# B&R Automation Studio project Soiled_PLC (part 9)

### CAN.typ
```iecst
TYPE
	WET_CAN : 	STRUCT
		ControlSignals : USINT;
		ControlSignals2 : USINT;
		Category : UINT;
		Customer : UINT;
		Weight : UINT;
	END_STRUCT;
	DRY_CAN : 	STRUCT
		ControlSignals : USINT;
		ControlByte2 : USINT;
		Category : UDINT;
		Weight : UINT;
	END_STRUCT;
	DRY_CAN1 : 	STRUCT
		CustomerCode : UDINT;
		BatchCode : UDINT;
	END_STRUCT;
	DRYCAN_comm_typ : 	STRUCT
		ReadFrame : DRY_CAN;
		WriteFrame : DRY_CAN;
		WriteFrame1 : DRY_CAN1;
		EventRead : BOOL;
		EventWrite : BOOL;
		EventWrite1 : BOOL;
	END_STRUCT;
	CAN_Vars : 	STRUCT
		StrobeComplete : BOOL;
		BagReady : BOOL;
		BatchCode : UINT;
		Category : UDINT;
		Customer : UDINT;
		Destination : UINT;
		DropLoad : BOOL;
		DoubleLoad : BOOL;
		Drier1Loading : BOOL;
		Drier2Loading : BOOL;
		Drier1Unloading : BOOL;
		Drier2Unloading : BOOL;
		FaultNumber : USINT;
		Live : BOOL;
		LiveTime : UINT;
		LoadDropped : BOOL;
		LoadFinished : BOOL;
		MachineID : UINT;
		Program : UINT;
		PressShift : BOOL;
		ReadyToLoad : BOOL;
		SP1 : UINT;
		SP2 : UINT;
		SP3 : UINT;
		Transfer : BOOL;
		UnloadFinished : BOOL;
		Weight : UINT;
		BatchID : UDINT;
		Batch_QtyRemaining : UINT;
		LoadRecieved : BOOL;
		Unloading : BOOL;
		Batchpart : ARRAY[0..7]OF Batchpart_typ;
		Batchpart_wgt : ARRAY[0..9]OF UINT;
	END_STRUCT;
	Batchpart_typ : 	STRUCT
		Wgt : UINT;
		Customer : UDINT;
	END_STRUCT;
	Comm_typ : 	STRUCT
		StrobeComplete : BOOL;
		BagReady : BOOL;
		BatchCode : UINT;
		Category : UDINT;
		Customer : UDINT;
		Destination : UINT;
		DropLoad : BOOL;
		DoubleLoad : BOOL;
		Live : BOOL;
		LiveTime : UINT;
		LoadDropped : BOOL;
		LoadFinished : BOOL;
		Program : UINT;
		ReadyToLoad : BOOL;
		UnloadFinished : BOOL;
		Weight : UINT;
		BatchID : UDINT;
		Batch_QtyRemaining : UINT;
		LoadRecieved : BOOL;
		Unloading : BOOL;
		Batchpart : ARRAY[0..7]OF Batchpart_typ;
		Batchpart_wgt : ARRAY[0..9]OF UINT;
		Count : UINT;
		Bid : UDINT; (**Internal use only pass bid ID>*)
		TimeStamp : DATE_AND_TIME; (**Internal use only*)
		Transfer : BOOL;
	END_STRUCT;
END_TYPE
```

### Program Logical/Sequences/200ms/CAN/can (IEC, version 2.00.0) - *DRY CAN

#### can.var
```iecst
VAR RETAIN
	CAN_enable : BOOL;
END_VAR
VAR
	CANdftab_01 : CANdftab;
	CANOK : BOOL;
	CANopen_01 : CANopen;
	CANrwtab_01 : CANrwtab;
	data_adr : UDINT;
	DOInfo : DatObjInfo;
	error_var : UDINT;
	LastError : UINT;
	n : UINT;
	MAX_CAN_CONNS : UINT;
	CAN_DRY_Send : ARRAY[0..19] OF DRYCAN_comm_typ;
	x : UINT;
END_VAR
```

#### can.ab
```automation-basic
;CAN Bus data exchange with CBW

;--------------------------------------------------------
;Version 1.00 02/11/2009 D.J. First Issue
;Version 2.00 22/011/2011 D.J. Weight Calculation now here
;--------------------------------------------------------

PROGRAM _INIT

CAN_enable = 1
MAX_CAN_CONNS = 6

LOOP n = 1 TO MAX_CAN_CONNS DO
	CAN_DRY_Send[n].EventRead = 0
	CAN_DRY_Send[n].EventWrite = 0
	CAN_DRY_Send[n].EventWrite1 = 0
ENDLOOP

CANopen_01.enable		= CAN_enable
CANopen_01.baud_rate	= 25					;Define baud rate - 250 kbit/s
CANopen_01.cob_anz		= 100      				;Define number of link objects
CANopen_01.error_adr	= ADR(error_var)		;Define address for error output
CANopen_01.device		= ADR("SS1.IF2")	    ;Define number of device
CANopen_01.info			= 0

CANopen_01 FUB CANopen()						;Initiate CANopen

IF CANopen_01.status=0 THEN						;Check error level

	DOInfo.enable = 1
	DOInfo.pName  = "can_cmd"

	DOInfo FUB DatObjInfo()

	IF (DOInfo.status = 0) THEN

		data_adr					= DOInfo.pDatObjMem
		CANdftab_01.enable			= 1
		CANdftab_01.us_ident 		= CANopen_01.us_ident	;Set us_id
		CANdftab_01.table_adr		= data_adr				;Define address of data object
		CANdftab_01.tab_num			= UINT(DOInfo.len / 72)	;Define number of values

		CANdftab_01 FUB CANdftab()    						;Initiate CANdftab

		IF CANdftab_01.status = 0 THEN
			LOOP n = 1 TO MAX_CAN_CONNS DO
				CAN_DRY_Send[n].WriteFrame.ControlSignals.0 = 1 // Set CAN Live
			ENDLOOP
			CANOK = TRUE
		ENDIF
	ENDIF
ENDIF

END_PROGRAM

PROGRAM _CYCLIC

IF CANOK THEN

	;----------------
	;Set Write values
	;---------------
	LOOP n = 3 TO MAX_CAN_CONNS DO
		CAN_DRY_Send[n].WriteFrame.ControlSignals.1 = CAN[n].BagReady
		CAN_DRY_Send[n].WriteFrame.Category			= CAN[n].Category
		CAN_DRY_Send[n].WriteFrame.Weight			= CAN[n].Weight
		CAN_DRY_Send[n].WriteFrame1.CustomerCode	= CAN[n].Customer
		CAN_DRY_Send[n].WriteFrame1.BatchCode		= CAN[n].BatchID
		CAN_DRY_Send[n].EventWrite = 1
		CAN_DRY_Send[n].EventWrite1 = 1
	ENDLOOP

	;-----------------
	;Service CAN table
	;-----------------
	IF CANdftab_01.status=0 THEN						(*check error level*)
		CANrwtab_01.enable		= 1
		CANrwtab_01.tab_ident	= CANdftab_01.tab_ident (*define tab_id*)
		CANrwtab_01 FUB CANrwtab()						(*initiate CANrwtab*)
		LastError = CANrwtab_01.status
	ENDIF

;	;----------------------------------
		;	;Check for incomming data from CBW1
		;	;----------------------------------
	LOOP n = 3 TO MAX_CAN_CONNS DO

		IF (CAN_DRY_Send[n].EventRead > 0)THEN
			CAN_DRY_Send[n].EventRead = 0

			CAN[n].Live 		  = CAN_DRY_Send[n].ReadFrame.ControlSignals.0
			CAN[n].DropLoad 	  = CAN_DRY_Send[n].ReadFrame.ControlSignals.1
			CAN[n].LoadDropped    = CAN_DRY_Send[n].ReadFrame.ControlSignals.2
			IF CAN[n].Live THEN
				CAN[n].LiveTime = 50	;5 seconds
			ENDIF
		ENDIF
		;~~~~~~~~~~~~~~~~~~~~~~~~~~~~~~~~~~~~~~~~~~~~~~~~
		;-------------------
		;CAN Live / Presence
		;-------------------
		IF (CAN[n].LiveTime > 0) THEN
			CAN[n].LiveTime = (CAN[n].LiveTime - 1)
		ENDIF
		CAN[n].Live = (CAN[n].LiveTime <> 0)

	ENDLOOP

ENDIF
END_PROGRAM
```

### Data object Logical/Sequences/200ms/CAN/can_cmd_wet (Simple) - *WET CAN I

#### can_cmd.dat
```
;-----------------
;CAN Command Table
;-----------------

;         1234567890123456789012345678901   1234567890123456789012345678901
00000121,"CAN_Drv2:ReadFrame1            ","CAN_Drv2:EventRead1            ",$00000000
00000120,"CAN_Drv2:WriteFrame1           ","CAN_Drv2:EventWrite1           ",$00000001

00000131,"CAN_Drv2:ReadFrame2            ","CAN_Drv2:EventRead2            ",$00000000
00000130,"CAN_Drv2:WriteFrame2           ","CAN_Drv2:EventWrite2           ",$00000001

; CAN ADR  Variable Name 31 Chrs             Event Variable 31 Chrs           Read = 0 Write = 1
```

- Program Logical/Sequences/200ms/CAN/CAN_Live (IEC) - * CAN Live status 1-32 to TrackView (no source held here)

### Data object Logical/Sequences/200ms/CAN/can1_cmd (Simple, version 1.00.0) - * Powertrans 1 & 2

#### can_cmd.dat
```
;-----------------
;CAN Command Table
;-----------------

;         1234567890123456789012345678901   1234567890123456789012345678901
00000251,"can_drv1:ReadFrame1            ","can_drv1:EventRead1            ",$00000000
00000241,"can_drv1:WriteFrame1           ","can_drv1:EventWrite1           ",$00000001
;123456789123456789123456789123456789123456789123456789123456789123456789
;00000121,"can_drv1:ReadFrame2            ","can_drv1:EventRead2            ",$00000000
;00000120,"can_drv1:WriteFrame2           ","can_drv1:EventWrite2           ",$00000001

;00000141,"ReadFrame3                     ","EventRead3                     ",$00000000
;00000140,"WriteFrame3                    ","EventWrite3                    ",$00000001
;   |          |                                 |                               |
; CAN ADR  Variable Name 31 Chrs             Event Variable 31 Chrs           Read = 0 Write = 1
```

### Program Logical/Sequences/200ms/CAN/can_drv1 (IEC) - * PowerTrans 1 SDC2

#### can_drv2.var
```iecst
VAR RETAIN
	CAN_enable : BOOL;
	ReadFrame1 : WET_CAN;
	EventRead1 : BOOL;
	EventWrite1 : BOOL;
	LastError : UINT;
	n : UINT;
	CANOK : BOOL;
	WriteFrame1 : WET_CAN;
	EventWrite2 : BOOL;
END_VAR
VAR
	ReadFrame2 : WET_CAN;
	EventRead2 : BOOL;
	WriteFrame2 : WET_CAN;
	CANopen_01 : CANopen;
	DOInfo : DatObjInfo;
	CANdftab_01 : CANdftab;
	error_var : UDINT;
	data_adr : UDINT;
	CANrwtab_01 : CANrwtab;
	TEST : BOOL;
END_VAR
```

#### can_drv2Cyclic.ab
```automation-basic
PROGRAM _CYCLIC
;----------------------------------------
;Version 1.00 08/02/2005 D.J. First Issue
;----------------------------------------

IF CANOK THEN

	;----------------
	;Set Write values
	;----------------

	;Powertrans 1
	IF CAN[1].BagReady THEN
		WriteFrame1.ControlSignals = BIT_SET(WriteFrame1.ControlSignals, 1)
	ELSE
		WriteFrame1.ControlSignals = BIT_CLR(WriteFrame1.ControlSignals, 1)
	ENDIF
   IF CAN[1].LoadFinished = TRUE THEN
			WriteFrame1.ControlSignals = BIT_SET(WriteFrame1.ControlSignals, 2)
	ELSE
			WriteFrame1.ControlSignals = BIT_CLR(WriteFrame1.ControlSignals, 2)
	ENDIF
	//WriteFrame1.Destination = 0
	WriteFrame1.Category 	= UINT(CAN[1].Category)
	WriteFrame1.Customer    = UINT(CAN[1].Customer)
	WriteFrame1.Weight      = CAN[1].Weight

	;Write to Machine1
	EventWrite1 = TRUE

	;Powertrans 2
	IF CAN[2].BagReady THEN
		WriteFrame2.ControlSignals = BIT_SET(WriteFrame2.ControlSignals, 1)
	ELSE
		WriteFrame2.ControlSignals = BIT_CLR(WriteFrame2.ControlSignals, 1)
	ENDIF
	;IF CAN[2].DoubleLoad THEN
	;	WriteFrame2.ControlSignals = BIT_SET(WriteFrame2.ControlSignals, 2)
	;ELSE
	;	WriteFrame2.ControlSignals = BIT_CLR(WriteFrame2.ControlSignals, 2)
	;ENDIF
	//WriteFrame2.Destination = 0
	WriteFrame2.Category 	= UINT(CAN[2].Category)
	WriteFrame2.Customer    = UINT(CAN[2].Customer)
	WriteFrame2.Weight      = CAN[2].Weight

	;Write to Machine2
	EventWrite2 = TRUE

	;-----------------
	;Service CAN table
	;-----------------

	IF CANdftab_01.status=0 THEN						(*check error level*)
		CANrwtab_01.enable		= 1
		CANrwtab_01.tab_ident	= CANdftab_01.tab_ident (*define tab_id*)
		CANrwtab_01 FUB CANrwtab()						(*initiate CANrwtab*)
		LastError = CANrwtab_01.status
	ENDIF

	;----------------------------------
	;Check for incomming data from CBW1
	;----------------------------------

	;Powertrans 1
	IF EventRead1 THEN

		EventRead1 = FALSE

		CAN[1].Live 		  = BIT_TST(ReadFrame1.ControlSignals,0)
		CAN[1].ReadyToLoad 	  = BIT_TST(ReadFrame1.ControlSignals,1)
        CAN[1].DropLoad           =  BIT_TST(ReadFrame1.ControlSignals,2)
		CAN[1].LoadDropped    = BIT_TST(ReadFrame1.ControlSignals,3)

		IF CAN[1].Live THEN
			CAN[1].LiveTime = 50	;5 seconds
		ENDIF

	ENDIF

	;----------------------------------
	;Check for incomming data from CBW2
	;----------------------------------

	;Powertrans 2
	IF EventRead2 THEN

		EventRead2 = FALSE

		CAN[2].Live 		  = BIT_TST(ReadFrame2.ControlSignals,0)
		CAN[2].DropLoad 	  = BIT_TST(ReadFrame2.ControlSignals,1)
		CAN[2].LoadDropped    = BIT_TST(ReadFrame2.ControlSignals,2)

		IF CAN[2].Live THEN
			CAN[2].LiveTime = 50	;5 seconds
		ENDIF

	ENDIF

	;-------------------
	;CAN Live / Presence
	;-------------------

	LOOP n = 1 TO 2 DO

		IF (CAN[n].LiveTime > 0) THEN
			CAN[n].LiveTime = (CAN[n].LiveTime - 1)
		ENDIF

		CAN[n].Live = (CAN[n].LiveTime <> 0)

	ENDLOOP

ENDIF
END_PROGRAM
```

#### can_drv2Init.ab
```automation-basic
PROGRAM _INIT
	(* init program *)

CAN_enable = 1
EventWrite1 = 0									;Reset CAN data table WRITE event
EventRead1 = 0  								;Reset CAN data table READ event
;EventWrite2 = 0								;Reset CAN data table WRITE event
;EventRead2 = 0  								;Reset CAN data table READ event
;EventWrite3 = 0								;Reset CAN data table WRITE event
;EventRead3 = 0  							    ;Reset CAN data table READ event

CANopen_01.enable		= CAN_enable
CANopen_01.baud_rate	= 25					;Define baud rate - 250 kbit/s
CANopen_01.cob_anz		= 100      				;Define number of link objects
CANopen_01.error_adr	= ADR(error_var)		;Define address for error output
CANopen_01.device		= ADR("SS1.IF1")	;Define number of device
CANopen_01.info			= 0

CANopen_01 FUB CANopen()						;Initiate CANopen

IF CANopen_01.status=0 THEN						;Check error level

	DOInfo.enable = 1
	DOInfo.pName  = "can1_cmd"

	DOInfo FUB DatObjInfo()

	IF (DOInfo.status = 0) THEN

		data_adr					= DOInfo.pDatObjMem
		CANdftab_01.enable			= 1
		CANdftab_01.us_ident 		= CANopen_01.us_ident	;Set us_id
		CANdftab_01.table_adr		= data_adr				;Define address of data object
		CANdftab_01.tab_num			= UINT(DOInfo.len / 72)	;Define number of values

		CANdftab_01 FUB CANdftab()    						;Initiate CANdftab

		IF CANdftab_01.status = 0 THEN
			WriteFrame1.ControlSignals = BIT_SET(WriteFrame1.ControlSignals,0);Set Live Signal
			WriteFrame2.ControlSignals = BIT_SET(WriteFrame2.ControlSignals,0)
			;WriteFrame3.ControlSignals = BIT_SET(WriteFrame3.ControlSignals,0)
			CANOK = TRUE
		ENDIF

	ENDIF

ENDIF
END_PROGRAM
```

### Program Logical/Sequences/200ms/CAN/can_drv2 (IEC, version 1.00.0) - * PowerTrans 1 SDC2

#### can_drv2Cyclic.ab
```automation-basic
PROGRAM _CYCLIC
;----------------------------------------
;Version 1.00 08/02/2005 D.J. First Issue
;----------------------------------------

IF CANOK THEN

	;----------------
	;Set Write values
	;----------------

	;Powertrans 1
	IF CAN[2].BagReady THEN
		WriteFrame2.ControlSignals = BIT_SET(WriteFrame2.ControlSignals, 1)
	ELSE
		WriteFrame2.ControlSignals = BIT_CLR(WriteFrame2.ControlSignals, 1)
	ENDIF
 IF CAN[2].LoadFinished = TRUE THEN
			WriteFrame2.ControlSignals = BIT_SET(WriteFrame2.ControlSignals, 2)
	ELSE
			WriteFrame2.ControlSignals = BIT_CLR(WriteFrame2.ControlSignals, 2)
	ENDIF
	//WriteFrame1.Destination = 0
	WriteFrame2.Category 	= UINT(CAN[2].Category)
	WriteFrame2.Customer    = UINT(CAN[2].Customer)
	WriteFrame2.Weight      = CAN[2].Weight

	;Write to Machine1
	EventWrite2 = TRUE

	//WriteFrame2.Destination = 0
	WriteFrame2.Category 	= UINT(CAN[2].Category)
	WriteFrame2.Customer    = UINT(CAN[2].Customer)
	WriteFrame2.Weight      = CAN[2].Weight

	;Write to Machine2
	EventWrite2 = TRUE

	;-----------------
	;Service CAN table
	;-----------------

	IF CANdftab_01.status=0 THEN						(*check error level*)
		CANrwtab_01.enable		= 1
		CANrwtab_01.tab_ident	= CANdftab_01.tab_ident (*define tab_id*)
		CANrwtab_01 FUB CANrwtab()						(*initiate CANrwtab*)
		LastError = CANrwtab_01.status
	ENDIF

	;----------------------------------
	;Check for incomming data from CBW1
	;----------------------------------

	;Powertrans 1
	IF EventRead2 THEN

		EventRead2 = FALSE

		CAN[2].Live 		          = BIT_TST(ReadFrame2.ControlSignals,0)
		CAN[2].ReadyToLoad	  = BIT_TST(ReadFrame2.ControlSignals,1)
		CAN[2].DropLoad          = BIT_TST(ReadFrame2.ControlSignals,2)
		CAN[2].LoadDropped    = BIT_TST(ReadFrame2.ControlSignals,3)

		IF CAN[2].Live THEN
			CAN[2].LiveTime = 50	;5 seconds
		ENDIF

	ENDIF

	;----------------------------------
	;Check for incomming data from CBW2
	;----------------------------------

	;-------------------
	;CAN Live / Presence
	;-------------------

	LOOP n = 1 TO 2 DO

		IF (CAN[n].LiveTime > 0) THEN
			CAN[n].LiveTime = (CAN[n].LiveTime - 1)
		ENDIF

		CAN[n].Live = (CAN[n].LiveTime <> 0)

	ENDLOOP

ENDIF
END_PROGRAM
```

#### can_drv2Init.ab
```automation-basic
PROGRAM _INIT
	(* init program *)

CAN_enable = 1
EventWrite1 = 0									;Reset CAN data table WRITE event
EventRead1 = 0  								;Reset CAN data table READ event
;EventWrite2 = 0								;Reset CAN data table WRITE event
;EventRead2 = 0  								;Reset CAN data table READ event
;EventWrite3 = 0								;Reset CAN data table WRITE event
;EventRead3 = 0  							    ;Reset CAN data table READ event

CANopen_01.enable		= CAN_enable
CANopen_01.baud_rate	= 25					;Define baud rate - 250 kbit/s
CANopen_01.cob_anz		= 100      				;Define number of link objects
CANopen_01.error_adr	= ADR(error_var)		;Define address for error output
CANopen_01.device		= ADR("SS1.IF2")	;Define number of device
CANopen_01.info			= 0

CANopen_01 FUB CANopen()						;Initiate CANopen

IF CANopen_01.status=0 THEN						;Check error level

	DOInfo.enable = 1
	DOInfo.pName  = "can2_cmd"

	DOInfo FUB DatObjInfo()

	IF (DOInfo.status = 0) THEN

		data_adr					= DOInfo.pDatObjMem
		CANdftab_01.enable			= 1
		CANdftab_01.us_ident 		= CANopen_01.us_ident	;Set us_id
		CANdftab_01.table_adr		= data_adr				;Define address of data object
		CANdftab_01.tab_num			= UINT(DOInfo.len / 72)	;Define number of values

		CANdftab_01 FUB CANdftab()    						;Initiate CANdftab

		IF CANdftab_01.status = 0 THEN
			WriteFrame1.ControlSignals = BIT_SET(WriteFrame1.ControlSignals,0);Set Live Signal
			WriteFrame2.ControlSignals = BIT_SET(WriteFrame2.ControlSignals,0)
			;WriteFrame3.ControlSignals = BIT_SET(WriteFrame3.ControlSignals,0)
			CANOK = TRUE
		ENDIF

	ENDIF

ENDIF
END_PROGRAM
```

### Program Logical/Sequences/200ms/CAN/can_dis (IEC)

#### can_dis.var
```iecst
VAR RETAIN
	CAN_enable : BOOL;
	LastError : UINT;
	n : UINT;
	CANOK : BOOL;
END_VAR
VAR
	CANopen_01 : CANopen;
	DOInfo : DatObjInfo;
	CANdftab_01 : CANdftab;
	error_var : UDINT;
	data_adr : UDINT;
	CANrwtab_01 : CANrwtab;
	DisplayWrite1 : BOOL;
	DisplayRead1 : BOOL;
	DisplayCat : ARRAY[0..32] OF USINT;
	DisplayWgt : ARRAY[0..16] OF UINT;
	DisplayCus : ARRAY[0..32] OF USINT;
	Display : ARRAY[0..87] OF UINT;
	Data : WriteDisplay;
	Reply : USINT;
	DisplayRXFrame5 : ReadDisplay;
	DisplayRXFrame4 : ReadDisplay;
	DisplayWrite4 : BOOL;
	DisplayTXFrame1 : WriteDisplay;
	DisplayWrite5 : BOOL;
	DisplayTXFrame2 : WriteDisplay;
	x : UINT;
	DisplayWrite6 : BOOL;
	DisplayTXFrame3 : WriteDisplay;
	DisplayRead2 : BOOL;
	DisplayTXFrame4 : WriteDisplay;
	DisplayRead3 : BOOL;
	DisplayTXFrame5 : WriteDisplay;
	Dummy : UINT;
	DisplayRead4 : BOOL;
	DisplayRXFrame1 : ReadDisplay;
	DisplayTXFrame6 : WriteDisplay;
	DisplayRead5 : BOOL;
	DisplayRXFrame2 : ReadDisplay;
	DisplayRead6 : BOOL;
	DisplayRXFrame3 : ReadDisplay;
	StepsRequired : UINT;
	DisplayChrs : UINT;
	DisplayRXFrame6 : ReadDisplay;
	STEP : UINT;
	Wgt1s : UINT;
	DisplayWrite2 : BOOL;
	DisplayWrite3 : BOOL;
	Wgt10s : UINT;
	m : UINT;
	DisplayTXFrame7 : WriteDisplay;
	DisplayTXFrame8 : WriteDisplay;
	DisplayTXFrame9 : WriteDisplay;
	DisplayTXFrame10 : WriteDisplay;
	DisplayTXFrame11 : WriteDisplay;
	DisplayTXFrame12 : WriteDisplay;
	DisplayTXFrame13 : WriteDisplay;
	DisplayWrite7 : BOOL;
	DisplayWrite8 : BOOL;
	DisplayWrite9 : BOOL;
	DisplayWrite10 : BOOL;
	DisplayWrite11 : BOOL;
	DisplayWrite12 : BOOL;
	DisplayWrite13 : BOOL;
	DisplayWrite14 : BOOL;
	DisplayWrite15 : BOOL;
	DisplayWrite16 : BOOL;
	DisplayRead7 : BOOL;
	DisplayRead8 : BOOL;
	DisplayRead9 : BOOL;
	DisplayRead10 : BOOL;
	DisplayRead11 : BOOL;
	DisplayRead12 : BOOL;
	DisplayRead13 : BOOL;
	DisplayRead14 : BOOL;
	DisplayRead15 : BOOL;
	DisplayRead16 : BOOL;
	DisplayRXFrame7 : ReadDisplay;
	DisplayRXFrame8 : ReadDisplay;
	DisplayRXFrame9 : ReadDisplay;
	DisplayRXFrame10 : ReadDisplay;
	DisplayRXFrame11 : ReadDisplay;
	DisplayRXFrame12 : ReadDisplay;
	DisplayRXFrame13 : ReadDisplay;
	DisplayRXFrame14 : ReadDisplay;
	DisplayRXFrame15 : ReadDisplay;
	DisplayRXFrame16 : ReadDisplay;
	DisplayTXFrame14 : WriteDisplay;
	DisplayTXFrame15 : WriteDisplay;
	DisplayTXFrame16 : WriteDisplay;
	CatName : ARRAY[0..32] OF UINT;
	CusName : ARRAY[0..32] OF UINT;
END_VAR
```

#### can_disCyclic.ab
```automation-basic
PROGRAM _CYCLIC
;-----------------------------------------
;Revision 1.00 18/02/2002 D.J. First Issue
;-----------------------------------------

;2 * 20 or 2 * 40 chr VFD display

;Set D register where text for display is set E register for weight
DisplayChrs		= 80

;LOOP m = 1 TO 7 DO//16 DO
;
;
;	;memcpy(ADR(DisplayCat[m]),ADR(zzGetNamesData[m].CatName),16)
;;	memcpy(ADR(DisplayCus[m]),ADR(zzGetNamesData[m].CusName),16)
;
;ENDLOOP

LOOP x = 1 TO 7 DO//16 DO
	memcpy(ADR(DisplayCat[1]),ADR(zzGetNamesData[x].CatName),32);
	memcpy(ADR(DisplayCus[1]),ADR(zzGetNamesData[x].CusName),32)
	//Convert string to Wstring
	LOOP m = 1 TO 32 DO
		CatName[m] = UINT(DisplayCat[m])
		CusName[m] = UINT(DisplayCus[m])
	ENDLOOP

	DisplayWgt[x] = Bag[200 + x].Wgt

	memset(ADR(Display[0]) ,32,SIZEOF (Display))

	memcpy(ADR(Display[0]),ADR(CatName[1]),32)
	memcpy(ADR(Display[44]),ADR(CusName[1]),32)

	;As the weight value is a INT put into a UINT -0.1 = 65535
	;Display only if less than 500kg
	IF (DisplayWgt[x] < 5000) THEN
		DIS4(DisplayWgt[x],TRUE,Dummy,Wgt1s,Wgt10s,Dummy)
	ELSE
		Wgt1s 	= 0
		Wgt10s 	= 0
	ENDIF

	;Add Weight and goto next line
	Display[35] = $20 ;Space
	Display[36] = (48 + USINT(Wgt10s))
	Display[37] = (48 + USINT(Wgt1s))
	Display[38] = $6B 	;k
	Display[39] = $67 	;g
	Display[40] = $A	;Line Feed
	Display[41] = $D	;Carriage Return
	Display[42] = 0
	Display[43] = 0

	;Display[78] = $44	;D
	;Display[79] = $55	;U
	;Display[80] = $43	;C
	;Display[81] = $4B	;K
	;Display[82] = $45	;E
	;Display[83] = $52	;R

	;Cursor Off and Home
	IF (STEP = 0) THEN
		n = 0
		Data.Data[0] = $9B
		Data.Data[1] = $6C
		Data.Data[2] = $9B
		Data.Data[3] = $48
		Data.Data[4] = 0
		Data.Data[5] = 0
		Data.Data[6] = 0
		Data.Data[7] = 0
	ENDIF

	;Write text to the Display
	IF (STEP > 0) THEN
		Data.Data[0] = USINT(Display[0 + n])
		Data.Data[1] = USINT(Display[1 + n])
		Data.Data[2] = USINT(Display[2 + n])
		Data.Data[3] = USINT(Display[3 + n])
		Data.Data[4] = USINT(Display[4 + n])
		Data.Data[5] = USINT(Display[5 + n])
		Data.Data[6] = USINT(Display[6 + n])
		Data.Data[7] = USINT(Display[7 + n])
	ENDIF

	;Write to the CAN Frame For the Current Display
	IF (x = 1) THEN
		DisplayTXFrame1 = Data
	ELSE IF (x = 2) THEN
		DisplayTXFrame2 = Data
	ELSE IF (x = 3) THEN
		DisplayTXFrame3 = Data
	ELSE IF (x = 4) THEN
		DisplayTXFrame4 = Data
	ELSE IF (x = 5) THEN
		DisplayTXFrame5 = Data
	ELSE IF (x = 6) THEN
		DisplayTXFrame6 = Data
	ELSE IF (x = 7) THEN
		DisplayTXFrame7 = Data
	ELSE IF (x = 8) THEN
		DisplayTXFrame8 = Data
	ELSE IF (x = 9) THEN
		DisplayTXFrame9 = Data
	ELSE IF (x = 10) THEN
		DisplayTXFrame10 = Data
	ELSE IF (x = 11) THEN
		DisplayTXFrame11 = Data
	ELSE IF (x = 12) THEN
		DisplayTXFrame12 = Data
	ELSE IF (x = 13) THEN
		DisplayTXFrame13 = Data
	ELSE IF (x = 14) THEN
		DisplayTXFrame14 = Data
	ELSE IF (x = 15) THEN
		DisplayTXFrame15 = Data
	ELSE IF (x = 16) THEN
		DisplayTXFrame16 = Data
	ENDIF

ENDLOOP

IF (STEP > 0) THEN
	n = n + 8
ENDIF

STEP = STEP + 1

StepsRequired = ((DisplayChrs / 8) + 1) ;Steps = Total Chrs / 8 + 1
IF STEP > StepsRequired THEN
	STEP = 0
ENDIF

IF CANOK THEN

	;------------------------------------------------------
	;Configure the CAN write to CBW1 SDC1
	;------------------------------------------------------

	;Write to Displays
	DisplayWrite1 = TRUE
	;DisplayWrite2 = TRUE
	DisplayWrite3 = TRUE
	;DisplayWrite4 = TRUE
	DisplayWrite5 = TRUE
	;DisplayWrite6 = TRUE
	DisplayWrite7 = TRUE
	;DisplayWrite8 = TRUE
	;DisplayWrite9 = TRUE
	;DisplayWrite10 = TRUE
	;DisplayWrite11 = TRUE
	;DisplayWrite12 = TRUE
	;DisplayWrite13 = TRUE
	;DisplayWrite14 = TRUE
	;DisplayWrite15 = TRUE
	;DisplayWrite16 = TRUE

	;------------------------
	;Service CAN table
	;------------------------

	IF CANdftab_01.status=0 THEN						(*check error level*)
		CANrwtab_01.enable		= 1
		CANrwtab_01.tab_ident	= CANdftab_01.tab_ident (*define tab_id*)
		CANrwtab_01 FUB CANrwtab()						(*initiate CANrwtab*)
		LastError = CANrwtab_01.status
	ENDIF

	;-----------------
	;Read Display Data
	;-----------------
	IF DisplayRead1 THEN
		DisplayRead1 = FALSE
		Reply = DisplayRXFrame1.Data[1]
	ENDIF
	IF DisplayRead2 THEN
		DisplayRead2 = FALSE
		Reply = DisplayRXFrame2.Data[1]
	ENDIF
	IF DisplayRead3 THEN
		DisplayRead3 = FALSE
		Reply = DisplayRXFrame3.Data[1]
	ENDIF
	IF DisplayRead4 THEN
		DisplayRead4 = FALSE
		Reply = DisplayRXFrame4.Data[1]
	ENDIF
	IF DisplayRead5 THEN
		DisplayRead5 = FALSE
		Reply = DisplayRXFrame5.Data[1]
	ENDIF
	IF DisplayRead6 THEN
		DisplayRead6 = FALSE
		Reply = DisplayRXFrame6.Data[1]
	ENDIF
	IF DisplayRead7 THEN
		DisplayRead7 = FALSE
		Reply = DisplayRXFrame7.Data[1]
	ENDIF
	IF DisplayRead8 THEN
		DisplayRead8 = FALSE
		Reply = DisplayRXFrame8.Data[1]
	ENDIF
	IF DisplayRead9 THEN
		DisplayRead9 = FALSE
		Reply = DisplayRXFrame9.Data[1]
	ENDIF
	IF DisplayRead10 THEN
		DisplayRead10 = FALSE
		Reply = DisplayRXFrame10.Data[1]
	ENDIF
	IF DisplayRead11 THEN
		DisplayRead11 = FALSE
		Reply = DisplayRXFrame11.Data[1]
	ENDIF
	IF DisplayRead12 THEN
		DisplayRead12 = FALSE
		Reply = DisplayRXFrame12.Data[1]
	ENDIF
	IF DisplayRead13 THEN
		DisplayRead13 = FALSE
		Reply = DisplayRXFrame13.Data[1]
	ENDIF
	IF DisplayRead14 THEN
		DisplayRead14 = FALSE
		Reply = DisplayRXFrame14.Data[1]
	ENDIF
	IF DisplayRead15 THEN
		DisplayRead15 = FALSE
		Reply = DisplayRXFrame15.Data[1]
	ENDIF
	IF DisplayRead16 THEN
		DisplayRead16 = FALSE
		Reply = DisplayRXFrame16.Data[1]
	ENDIF

ENDIF

END_PROGRAM
```

#### can_disInit.ab
```automation-basic
PROGRAM _INIT
	(* init program *)

CAN_enable = 1
DisplayWrite1 = 0								;Reset CAN data table WRITE event
DisplayRead1 = 0  								;Reset CAN data table READ event
;EventWrite2 = 0								;Reset CAN data table WRITE event
;EventRead2 = 0  								;Reset CAN data table READ event
;EventWrite3 = 0								;Reset CAN data table WRITE event
;EventRead3 = 0  							    ;Reset CAN data table READ event

CANopen_01.enable		= CAN_enable
CANopen_01.baud_rate	= 25					;Define baud rate - 250 kbit/s
CANopen_01.cob_anz		= 100      				;Define number of link objects
CANopen_01.error_adr	= ADR(error_var)		;Define address for error output
CANopen_01.device		= ADR("SS1.IF2")		;Define number of device
CANopen_01.info			= 0

CANopen_01 FUB CANopen()						;Initiate CANopen

IF CANopen_01.status=0 THEN						;Check error level

	DOInfo.enable = 1
	DOInfo.pName  = "disp_cmd"

	DOInfo FUB DatObjInfo()

	IF (DOInfo.status = 0) THEN

		data_adr					= DOInfo.pDatObjMem
		CANdftab_01.enable			= 1
		CANdftab_01.us_ident 		= CANopen_01.us_ident	;Set us_id
		CANdftab_01.table_adr		= data_adr				;Define address of data object
		CANdftab_01.tab_num			= UINT(DOInfo.len / 72)	;Define number of values

		CANdftab_01 FUB CANdftab()    						;Initiate CANdftab

		IF CANdftab_01.status = 0 THEN
			CANOK = TRUE
		ENDIF

	ENDIF

ENDIF
END_PROGRAM
```

### Data object Logical/Sequences/200ms/CAN/can2_cmd (Simple)

#### disp_cmd.dat
```
;-----------------
;CAN Command Table
;-----------------

;         1234567890123456789012345678901   1234567890123456789012345678901
;CAN Node 11
00000251,"can_drv2:ReadFrame2            ","can_drv2:EventRead2            ",$00000000
00000241,"can_drv2:WriteFrame2           ","can_drv2:EventWrite2           ",$00000001

;   |          |                                 |                               |
; CAN ADR  Variable Name 31 Chrs             Event Variable 31 Chrs           Read = 0 Write = 1
```

### Package Logical/Sequences/200ms/Reports - Reports Variables

### Reports.typ
```iecst
TYPE
	Report : 	STRUCT
		Cat : UDINT;
		Cus : UDINT;
		Mis : UDINT;
		Bid : UDINT;
		Ur2 : UDINT;
		Prg : UINT;
		Wgt : UINT;
		Cnt : UINT;
		Stn : UINT;
		Mcn : UINT;
		Dst : UINT;
		Ur1 : UINT;
		Act : UINT;
		Rkg : UINT;
		TimeStamp : DATE_AND_TIME;
	END_STRUCT;
END_TYPE
```

### Reports.var
```iecst
VAR RETAIN
	ReportBuffer : ARRAY[0..199] OF Report;
	ReportLoading : ARRAY[0..60] OF Report;
	ReportUnloading : ARRAY[0..10] OF Report;
END_VAR
```

### Program Logical/Sequences/200ms/Reports/zzReport (IEC, version 3.00.0) - * Reports to Master PC

#### zzreport.var
```iecst
VAR RETAIN
	ReportID : UDINT;
END_VAR
VAR
	n : UINT;
	ReportPointer : UINT;
	MaxReportBuffer : UINT;
	MaxReportLoading : UINT;
	MaxReportUnloading : UINT;
	TestUnloadingCat : UINT;
	AddUnloading : BOOL;
	AddRepport : BOOL;
	AddReport : BOOL;
	AddStn : UDINT;
	AddMcn : UDINT;
	AddMis : UDINT;
	AddBid : UDINT;
	AddCat : UDINT;
	AddCus : UDINT;
	AddWgt : UINT;
	AddAct : UINT;
	AddUr1 : UDINT;
	AddUr2 : UDINT;
	AddRkg : UDINT;
END_VAR
```

#### zzreport.ab
```automation-basic
PROGRAM _CYCLIC
	;Reports To Graphics  - No changes required!

	;--------------------------------------------------
	;Revision 1.00 19/01/2006 First Issue D.J.
	;Revision 2.00 24/06/2009 32Bit Version D.J.
	;Revision 3.00 09/11/2011 Added Mis (Batch ID) D.J.
	;--------------------------------------------------

	;ReportBuffer 0 used to clear report all Zero
	ReportBuffer[0].Cat = 0
	ReportBuffer[0].Cus = 0
	ReportBuffer[0].Mis = 0
	ReportBuffer[0].Bid = 0
	ReportBuffer[0].Wgt = 0
	ReportBuffer[0].Cnt = 0
	ReportBuffer[0].Stn = 0
	ReportBuffer[0].Mcn = 0
	ReportBuffer[0].Prg = 0
	ReportBuffer[0].Dst = 0

	;Report array sizes - see declerations
	MaxReportBuffer		= 198	;1 less than array allocation as Array 0 is used as Zero values
	MaxReportLoading 	= 59	;Normally at least MaxStations
	MaxReportUnloading 	= 9		;Normally at least MaxDischargers

	;Shuffle reports buffer
	ReportPointer		= 0 	;Reports Pointer

	LOOP n = 1 TO MaxReportBuffer DO

		IF ((ReportBuffer[n].Cat = 0) AND (n < MaxReportBuffer)) THEN
			ReportBuffer[n] 		= ReportBuffer[n + 1]
			ReportBuffer[n + 1] 	= ReportBuffer[0]
		ENDIF

		;Inc Reports Pointer
		IF (ReportBuffer[n].Cat > 0) THEN
			ReportPointer = (ReportPointer + 1)
		ENDIF

	ENDLOOP

	;Put loaded reports into reports buffer
	LOOP n = 1 TO MaxReportLoading DO
		IF ((ReportBuffer[ReportPointer + 1].Cat = 0) AND (ReportPointer < MaxReportBuffer)) THEN
			IF (ReportLoading[n].Cat > 0) THEN
				ReportBuffer[ReportPointer + 1] = ReportLoading[n]
				ReportLoading[n] 				= ReportBuffer[0]
				ReportPointer 					= (ReportPointer + 1)
			ENDIF
		ENDIF
	ENDLOOP

	;Put unloaded reports into reports buffer
	LOOP n = 1 TO MaxReportUnloading DO
		IF ((ReportBuffer[ReportPointer + 1].Cat = 0) AND (ReportPointer < MaxReportBuffer)) THEN
			IF ReportUnloading[n].Cat > 0 THEN
				ReportBuffer[ReportPointer + 1] = ReportUnloading[n]
				ReportUnloading[n] 				= ReportBuffer[0]
				ReportPointer 					= (ReportPointer + 1)
			ENDIF
		ENDIF
	ENDLOOP

	;Reports Read from Graphics D32[20]
	;Generate Unique Report ID
	IF (D32[20] = ReportID) THEN
		;Clear first report
		ReportBuffer[1] = ReportBuffer[0]
		;Inc Report ID
		ReportID = ReportID + 1
	ENDIF

	;Set Report ID to Valid Range
	IF ((ReportID < 1) OR (ReportID > 9999)) THEN
		ReportID = 1
	ENDIF

	;Make Report at front of Q ready for Graphics
	IF (ReportBuffer[1].Cat > 0) THEN	;Reports Waiting
		D32[1] = 1
	ELSE
		D32[1] = 0
	ENDIF
	D32[2] 	= ReportBuffer[1].Cus 			;D2 = Reports Customer
	D32[3] 	= ReportBuffer[1].Cat 			;D3 = Reports Category
	D32[4] 	= UDINT(ReportBuffer[1].Wgt) 	;D4 = Reports Weight
	D32[5] 	= UDINT(ReportBuffer[1].Cnt) 	;D5 = Reports Count
	D32[6] 	= UDINT(ReportBuffer[1].Stn) 	;D6 = Reports Station
	D32[7] 	= UDINT(ReportBuffer[1].Mcn) 	;D7 = Reports Machine
	D32[8] 	= ReportBuffer[1].Cat //UDINT(ReportBuffer[1].Prg)	;D8 = Reports Program (New)
	D32[9] 	= ReportBuffer[1].Bid			;D9 = Reports Bag ID
	D32[10] = ReportBuffer[1].Dst			;D10 = Reports Destination

	D32[13] = ReportBuffer[1].Mis			;D13 = Reports Mis Server (Batch ID)
	D32[14] = ReportBuffer[1].Act			;D14 = Reports Action - ie Release / Mix
	D32[15] = ReportBuffer[1].Ur1			;D15 = User 1
	D32[16] = ReportBuffer[1].Ur2			;D16 = User 2
	D32[17]	= ReportBuffer[1].Rkg			;D17 = Bag release weight

	D32[19] = ReportID

	;---------------
	;Reports testing
	;---------------

	;Add report
	IF (AddReport AND (Bag[1].Cat > 0)) THEN
		IF (ReportUnloading[1].Cat = 0) THEN
			ReportUnloading[1].Cat = AddCat				;Category
			ReportUnloading[1].Cus = AddCus				;Customer
			ReportUnloading[1].Wgt = UINT(AddWgt)				;Weight
			ReportUnloading[1].Cnt = 0					;Count
			ReportUnloading[1].Stn = UINT(AddStn)		;Station
			ReportUnloading[1].Mcn = UINT(AddMcn)		;Machine
			ReportUnloading[1].Mis = AddMis				;MIS ID
			ReportUnloading[1].Bid = AddBid
			ReportUnloading[1].Act = UINT(AddAct)
			ReportUnloading[1].Ur1 = UINT(AddUr1)
			ReportUnloading[1].Ur2 = AddUr2
			ReportUnloading[1].Rkg = UINT(AddRkg)
			;ReportUnloading[1].TimeStamp = myTimeStamp
			ReportUnloading[1].TimeStamp = CurrentTimestamp
	ENDIF
		AddReport = FALSE
	ENDIF
END_PROGRAM
```

### Program Logical/Sequences/200ms/zzAlarms (IEC, version 4.00.0) - Alarms - Messages and History

#### zzalarms.var
```iecst
VAR RETAIN
	I_CancelAlarm : BOOL;
END_VAR
VAR
	BuildD220 : UINT;
	AlmNumber : UINT;
	n : UINT;
	AlarmCount : UINT;
	CancelBeacon : BOOL;
	I_MotorOverload : BOOL;
	UnloadingAlarm : BOOL;
	I_InverterFault : BOOL;
	BeaconInList : BOOL;
	ConstKeep : UINT;
	I_SystemStopped : BOOL;
	AlarmOutput : BOOL;
	tmrAlmOutput : TON_10ms;
	I_SafetyHighLevel : BOOL;
	I_Safetyloading : BOOL;
	I_SafetyVC : ARRAY[0..2] OF BOOL;
	I_EStop : BOOL;
	CancelAlarm : BOOL;
	Y816 : BOOL;
	Siren : BOOL;
	SirenET : UDINT;
	KEV : UINT;
END_VAR
```

#### zzalarms.ab
```automation-basic
PROGRAM _CYCLIC
	(* cyclic program *)

;-----------------------------------------------
;Alarm Messages with Screen position and history
;-----------------------------------------------

;-----------------------------------------------------------------
;Version 1.00 - 08/12/2005 First Issue D.J.
;Version 2.00 - 17/10/2006 Added Alarm.Extra D.J.
;Version 3.00 - 23/04/2007 Added Constants to stop them being lost
;Version 4.00 - 01/12/2009 Changed to 200 from 100 Sequence Alarms
;-----------------------------------------------------------------

;Alarm Constnts
ConstKeep = almBagDataError
ConstKeep = almBagNotArrived
ConstKeep = almBagNotAtProx
ConstKeep = almBagNotReleased
ConstKeep = almBagNotSettled
ConstKeep = almBagNotShownOnScreen
ConstKeep = almBagOverWeight
ConstKeep = almCarriageMoveFault
ConstKeep = almClearingBeltPleaseWait
ConstKeep = almDestinationNotValid
ConstKeep = almEmergencyStop
ConstKeep = almGeneralSequence
ConstKeep = almInverterFault
ConstKeep = almLoadNotDropped
ConstKeep = almMotorOverload
ConstKeep = almNoAlarm
ConstKeep = almPhotocellBlocked
ConstKeep = almPhotocellNotMade
ConstKeep = almStationNotClosed
ConstKeep = almStationNotEmpty
ConstKeep = almSwitchFault
ConstKeep = almUldNoBag
ConstKeep = almUldProgFinished
ConstKeep = almSystemStopped

;Note - Sequence must set the following
;Alarm[x].on
;Alarm[x].Bag - for the bag position where the alarm will appear
;Alarm[x].Name - for the message that will be displayed use constants strating "alm"
;Alarn[x].Extra - Extra data for Graphics to use ie. Line number with fault on offgoing storage

I_CancelAlarm 	= FALSE ;X[4].X16
I_EStop 		= Std.EStop; OR Std.EStopLoading
I_MotorOverload = Std.MotorOverload OR Std.MotorOverloadLoading
I_SystemStopped = NOT Std.SafetyOn
I_InverterFault = FALSE ;(X[3].X03 OR X[3].X04 OR X[3].X05 OR X[3].X06)
;I_SafetyHighLevel	= Std.HaltSys
;I_Safetyloading		= Std.HaltSysLoading
;I_SafetyVC[1]		= Std.HaltSysVC[1]
;I_SafetyVC[2]		= Std.HaltSysVC[2]
;--------------
;Alarm Messages
;--------------

IF I_EStop THEN
	Alarm[200].On	= TRUE
	Alarm[200].Bag 	= 0
	Alarm[200].Name	= almEmergencyStop
ELSE IF I_MotorOverload THEN
	Alarm[200].On	= TRUE
	Alarm[200].Bag 	= 0
	;Alarm[200].Name	= almMotorOverload
	Alarm[200].Name	= KEV
ELSE IF I_SystemStopped THEN
	Alarm[200].On	= TRUE
	Alarm[200].Bag 	= 0
	Alarm[200].Name	= almSystemStopped
ELSE IF I_InverterFault THEN
	Alarm[200].On	= TRUE
	Alarm[200].Bag 	= 0
	Alarm[200].Name	= almInverterFault
ELSE
	Alarm[200].On	= FALSE
	Alarm[200].Bag 	= 0
	Alarm[200].Name	= almNoAlarm
ENDIF
LOOP n = 5 TO 9 DO
	Alarm[200 + n].On	= FALSE
	Alarm[200 + n].Bag 	= 0
	Alarm[200 + n].Name	= almNoAlarm
ENDLOOP
IF I_SafetyHighLevel THEN
	Alarm[205].On	= TRUE
	Alarm[205].Bag 	= 0
	Alarm[205].Name	= almSafetyHighLevel
ENDIF
IF I_Safetyloading THEN
	Alarm[206].On	= TRUE
	Alarm[206].Bag 	= 0
	Alarm[206].Name	= almSafetyLoading
ENDIF
IF I_SafetyVC[1] THEN	 ; Don't use VC alarms unless cust reqs as will
	Alarm[207].On	= TRUE
	Alarm[207].Bag 	= 0
	Alarm[207].Name	= almSafetyVC
	Alarm[207].Extra = 1
ENDIF
;IF I_SafetyVC[2] THEN
;	Alarm[208].On	= TRUE
;	Alarm[208].Bag 	= 0
;	Alarm[208].Name	= almSafetyVC
;	Alarm[208].Extra = 2
;ENDIF
;

;Shuffle the Alarms List

AlarmCount 		= 0
BeaconInList 	= FALSE

LOOP n = 1 TO 10 DO

	;If Alarm not on anymore the clear from the list
	AlmNumber = D[200 + n]
	IF NOT Alarm[AlmNumber].On THEN
		D[200 + n] = 0
		D[210 + n] = 0
	ENDIF

	;Shuffle the list down
	IF (D[200 + n] = 0) AND (D[201 + n] > 0) AND (n <> 10) THEN
		D[200 + n] = D[201 + n]
		D[210 + n] = D[211 + n]
		D[201 + n] = 0
		D[211 + n] = 0
	ENDIF

	;Set InList for any alarm in the list
	Alarm[D[200 + n]].InList = TRUE

	;Calculate total alarms in the list
	IF D[200 + n] > 0 THEN
		AlarmCount = AlarmCount + 1
	ENDIF

	;Is the alarm beacon required?
	IF Alarm[AlmNumber].On AND Alarm[AlmNumber].Beacon THEN
		BeaconInList = TRUE
	ENDIF

ENDLOOP

;Cancel the alarm beacon
IF I_CancelAlarm THEN
	CancelBeacon = TRUE
ENDIF

;Cancel the CancelAlarm beacon if no alarm in the list requires the beacon
IF NOT BeaconInList THEN
	CancelBeacon = FALSE
ENDIF

;Look at each sequence alarm and if not in list then add to list if space
LOOP n = 1 TO 209 DO

	;If alarm active and a code has been given and not in the list and history is clear then add
	IF ((AlarmCount < 10) AND Alarm[n].On AND NOT Alarm[n].InList AND ((D[221] = 0) OR (n > 200))) THEN

		;If name not set then set to general
		IF (Alarm[n].Name = 0) THEN
			Alarm[n].Name = almGeneralSequence
		ENDIF

		D[210] 			= n
		BuildD220		= LSL(Alarm[n].Extra,8)
		BuildD220 		= BuildD220 + Alarm[n].Name
		D[220] 			= BuildD220

		;New alarm found requiring the beacon
		IF Alarm[n].Beacon THEN
			CancelBeacon = FALSE
		ENDIF

		;Store to History - if not Unloading Alarm
		IF (n <= 200) THEN
			D[221] 			= n				;Alarm Number (Seq)
			D[222]			= Alarm[n].Name	;Alarm Name / Message
			D[223] 			= D[223] + 1	;Alarm ID
			D[224]			= Alarm[n].Extra;Alarm Extra Data
			IF D[223] > 32000 THEN
				D[223] = 1
			ENDIF
		ENDIF

		;Inc Total Alarms
		AlarmCount = AlarmCount + 1

	ENDIF

	;Cancel All InList's - will be checked on the next scan
	Alarm[n].InList = FALSE

ENDLOOP

;Show Alarm position on the screen
IF D[201] > 0 THEN
	D[0] = Alarm[D[201]].Bag
ELSE
	D[0] = 0
ENDIF
;Alarms 203> used for extra safety zones
UnloadingAlarm = (Alarm[201].On OR Alarm[202].On OR Alarm[203].On OR Alarm[204].On); OR Alarm[205].On OR Alarm[206].On OR Alarm[207].On OR Alarm[208].On)

;Alarm Output - Unloading Alarm cannot be cancelled
;Y[8].Y16 = ((BeaconInList AND NOT CancelBeacon) OR UnloadingAlarm)
;Y[8].Y15 = CancelAlarm
TON_10ms(Y[8].Y16,1200,Siren,SirenET)
;Y[8].Y14 = Siren
;Timed Alarm Output Horn or Beacon
AlarmOutput = BeaconInList; OR UnloadingAlarm)

tmrAlmOutput.IN = AlarmOutput
tmrAlmOutput.PT = 6000
tmrAlmOutput FUB TON_10ms()

IF tmrAlmOutput.Q THEN
	CancelBeacon = TRUE
ENDIF

;Y[3].Y01 = (AlarmOutput AND NOT CancelBeacon)

END_PROGRAM
```

- Program Logical/Sequences/200ms/zzTime (IEC) - * System running time (no source held here)

- Program Logical/Sequences/200ms/USB_Pmem (IEC, version 3.00.0) - * USB - Backup and Restore data (no source held here)

### Program Logical/Sequences/200ms/zzStn_Q (IEC, version 3.00.0)

#### zzstn_q.var
```iecst
VAR
	n : UINT;
	ValidWeight : BOOL;
	SP1Reached : BOOL;
	SP2Reached : BOOL;
	SP3Reached : BOOL;
	TestWeight : UINT;
	StnIntoQ : BOOL;
	StnsInQ : BOOL;
	PurgeStation : BOOL;
	StnsToPurge : BOOL;
	ManualRelease : BOOL;
	TestStation : UINT;
	z : UINT;
	Calibration : BOOL;
	ValidPurgeWeight : BOOL;
END_VAR
```

#### zzstn_q.ab
```automation-basic
PROGRAM _CYCLIC
 	(* cyclic program *)

;Sorting Stations Into Q with provision for Pushbutton into Q
;------------------------------------------------------------

;Set "AutoMaticRelease" in "zzconst"
;Nothing to change!

;--------------------------------------------------------------------
;Version 1.00 - 19/12/2005 D.J. First Issue
;Version 2.00 - 10/12/2009 D.J. Changed Setpoint Registers to D4000's
;Version 3.00 - 03/02/2011 D.J. Re-instated calibration stops release
;--------------------------------------------------------------------

StnsInQ 	= FALSE
;StnsToPurge = FALSE
Calibration = (D[998] > 0)

LOOP z = 1 TO Std.MaxWeighstations DO
;LOOP z = 8 TO 8 DO
	n = z

	;Force to Single station for testing / monitoring
	IF TestStation > 0 THEN
		n = TestStation
	ENDIF

	ManualRelease 	= (D[800 + n] = 1)
	PurgeStation	= (D[800 + n] = 2)

	;For testing force valid weight values
	IF TestWeight > 0 THEN
		Stn[n].Weight = TestWeight
	ENDIF

	;If Current weight is less than the Min Release Weight or SP2 is set below the Min Release Weight or SP3 is set below the Min Release Weight
	ValidWeight = ((Stn[n].Weight > Std.MinReleaseWeight) AND (D[4800 + n] > Std.MinReleaseWeight) AND  (D[4900 + n] > Std.MinReleaseWeight))

	;Zurich Test - min release at 10kg
	;ValidWeight = ((Stn[n].Weight > 100) AND (D[4800 + n] > 100) AND  (D[4900 + n] > 100))

	;SP1 Reached - Approaching Weight
	SP1Reached = (Stn[n].Weight > D[4700 + n])

	;SP2 Reached - At Release Weight
	SP2Reached = (Stn[n].Weight >= D[4800 + n])

	;SP3 Reached - Over Weight
	SP3Reached = (Stn[n].Weight > D[4900 + n])

	;Manual Release from TrackView
	IF ManualRelease THEN
		IF (ValidWeight AND (NOT SP3Reached)) THEN
			Stn[n].ManualRelease = TRUE
		ELSE IF (ValidWeight AND Std.EnableOverUnderRelease) THEN ;Enable Release KeySwitch
			Stn[n].ManualRelease = TRUE
		ENDIF
		D[800 + n] = 0 ;Cancel the Manual Release
		Stn[n].Purge = FALSE
	ENDIF

	ValidPurgeWeight = (Stn[n].Weight > Std.MinPurgeWeight)
	IF PurgeStation THEN
		Stn[n].Purge = ValidPurgeWeight AND NOT SP3Reached
		D[800 + n] = 0
	ENDIF

	;Enter Station into Q
	StnIntoQ = FALSE
	IF (Std.AutoMaticRelease AND SP2Reached AND ValidWeight AND (NOT SP3Reached)) THEN
		StnIntoQ = TRUE
	ELSE IF ((NOT Std.AutoMaticRelease) AND Stn[n].ReleaseButton AND SP2Reached AND ValidWeight AND (NOT SP3Reached)) THEN
		StnIntoQ = TRUE
	ELSE IF ((NOT Std.AutoMaticRelease) AND Stn[n].ReleaseButton AND Std.EnableOverUnderRelease AND ValidWeight) THEN
		StnIntoQ = TRUE
	ELSE IF (Stn[n].ManualRelease AND ValidWeight) THEN
		StnIntoQ = TRUE
	ELSE IF Stn[n].Purge THEN
		StnIntoQ = TRUE
	ELSE IF ((D[7900 + n] > 1) AND Stn[n].CloseFlap AND ValidWeight) THEN
		StnIntoQ = TRUE ;Once loading flap has been closed then keep in Q
	ENDIF

	IF Stn[n].ManualRelease AND NOT ValidWeight THEN
		Stn[n].ManualRelease = FALSE
	ENDIF
	;Don't allow station release if calibrating
	IF Calibration THEN
		StnIntoQ = FALSE
	ENDIF

	IF StnIntoQ THEN
		StnsInQ = TRUE
		IF (Stn[n].QTime < $7FFF) THEN ;Keep within Integer range for PC
			Stn[n].QTime = (Stn[n].QTime + 1)
		ENDIF
	ELSE
		Stn[n].QTime = 0
	ENDIF

	D[100 + n] = Stn[n].QTime ;Set the time in the Q for Use by PC

	Stn[n].SP1	= FALSE
	Stn[n].SP2	= FALSE
	Stn[n].SP3	= FALSE

	IF SP3Reached THEN
		Stn[n].SP3 = TRUE
	ELSE IF SP2Reached OR StnIntoQ THEN
		Stn[n].SP2 = TRUE
	ELSE IF SP1Reached THEN
		Stn[n].SP1 = TRUE
	ENDIF

ENDLOOP

Std.StnsInQ 	= StnsInQ
;Std.StnsToPurge = StnsToPurge

END_PROGRAM
```

### Program Logical/Sequences/200ms/zzWeigh (IEC, version 6.00.0) - * Station Weight Calculation and Calibration

#### zzweigh.var
```iecst
VAR RETAIN
	n : UINT;
	WeightUnits : DINT;
	StnHigh : UINT;
	StnLow : UINT;
	StnTestWgt : UINT;
	HighLow : UDINT;
	RawLow : DINT;
	StnRaw : ARRAY[0..99] OF UINT;
	NewLow : UINT;
	NewHigh : UINT;
END_VAR
VAR
	tstRaw : DINT;
	myRaw : DINT;
	myStnRaw : UINT;
	UseAI2744 : BOOL;
	FixCalibration : BOOL;
	Auto_ForceCalib : BOOL;
	Calib_Stn : UINT;
	Auto_Calib : enum_Calib;
	test1 : UINT;
	test2 : UINT;
	test3 : UINT;
	test4 : UINT;
	weighttest : BOOL;
END_VAR
```

#### zzweigh.ab
```automation-basic
PROGRAM _CYCLIC
	(* cyclic program *)

;---------------------------------------------------------------------------------------------
;Revision 1.00 01/05/2001 D.J. First Issu
;Revision 2.00 23/10/2002 D.J. WeightUnits changed to DINT (problem when raw values over 32767
;Revision 3.00 22/08/2006 D.J. Changed for AI261
;Revision 4.00 10/12/2009 D.J. Changed Calibration Storage Registers to D4400 etc.. AND AI2744
;Revision 5.00 09/08/2012 D.J. Changed Raw value to WeightRaw
;Revision 6.00 28/11/2012 D.J. Added Value Calibration values send to TrackView
;---------------------------------------------------------------------------------------------

;---------------------------------------------------------------------
;WeighStation Calibration and Weight Calculation - With AI261 & AI2744
;---------------------------------------------------------------------

UseAI2744 = FALSE ;Set PLC module type
IF Auto_ForceCalib THEN
	IF (Calib_Stn = 0) THEN
		Calib_Stn = 1
	ELSE IF Calib_Stn > Std.MaxWeighstations THEN
		Calib_Stn = 0
		Auto_ForceCalib = FALSE
	ENDIF
	D[940 + Calib_Stn] = 1
	CASE Auto_Calib OF
		ACTION Calib_Low:
			D[995] = Calib_Stn
			D[996] = 11
			AI261Raw[Calib_Stn] = 0
			Auto_Calib = Calib_High
		ENDACTION

		ACTION Calib_High:
			D[995] = Calib_Stn
			D[996] = 12
			D[997] = 200
			AI261Raw[Calib_Stn] = 20000
			Auto_Calib = Calib_Low
			INC Calib_Stn
		ENDACTION
	ENDCASE
ENDIF

;divide by 1000 (AI261) or 100 (AI2744) should give around 50 parts per kg and keep raw value within UINT
;Add 32000 to value to ensure always positive
LOOP n = 1 TO (Std.MaxWeighstations) DO
	;To view a particular stn then set tstRaw to the required stn

	IF tstRaw > 0 THEN
		myRaw = tstRaw ;WeightRaw[tstRaw]
	ELSE
;			IF (WeightRaw[n].Wgt_Channel_2 = 0) OR (WeightRaw[n].Wgt_Channel_2 = $007F_FFFF)THEN
;				myRaw = ABS(WeightRaw[n].Wgt_Channel_1)
;			ELSE
;				myRaw = ABS(((WeightRaw[n].Wgt_Channel_1 + WeightRaw[n].Wgt_Channel_2)/2))
;			ENDIF
		myRaw = AI261Raw[n]
	ENDIF

	myRaw = (myRaw - myRaw - myRaw)

	;Ensure raw value is within + 24bit if out of range + 32bit
	IF (myRaw = $7FFFFFFF) THEN
		myRaw = $FFFFFF
	ENDIF

	;Ensure raw value is within - 24bit if out of range - 32bit
	IF (myRaw = $80000001) THEN
		myRaw = $FF000001
	ENDIF
	;Convert raw to UINT the 3 least significant digits are removed
	IF UseAI2744 THEN
		myStnRaw = UINT((myRaw / 100) + 32000)
	ELSE
		myStnRaw = UINT((myRaw / 1000) + 32000)
	ENDIF
	StnRaw[n] = myStnRaw
ENDLOOP
StnRaw[1] = UINT(AI1223[1] + 32767)
StnRaw[2] = UINT(AI1223[2] + 32767)
StnRaw[3] = UINT(AI1223[3] + 32767)
StnRaw[4] = UINT(AI1223[4] + 32767)
StnRaw[5] = UINT(AI1223[5] + 32767)
StnRaw[6] = UINT(AI1223[6] + 32767)
StnRaw[7] = UINT(AI1223[7] + 32767)
StnRaw[8] = UINT(AI1223[8] + 32767)
StnRaw[9] = UINT(AI1223[9] + 32767)
StnRaw[10] = UINT(AI1223[10] + 32767)
StnRaw[11] = UINT(AI1223[11] + 32767)
StnRaw[12] = UINT(AI1223[12] + 32767)
StnRaw[13] = UINT(AI1223[13] + 32767)
StnRaw[14] = UINT(AI1223[14] + 32767)
StnRaw[15] = UINT(AI1223[15] + 32767)
StnRaw[16] = UINT(AI1223[16] + 32767)

LOOP n = 1 TO Std.MaxWeighstations DO

	StnLow 		= D[4400 + n]
	StnHigh 	= D[4500 + n]
	StnTestWgt 	= D[4600 + n]

	;Calibrate Low - From TrackView
	IF (D[995] = n) AND (D[996] = 11) THEN
		NewLow = StnRaw[n]
		IF (NewLow > 0) AND (NewLow < $FFFF) THEN
			D[4400 + n] = NewLow
		ENDIF
		D[996] = 0 ;Cancel the Cal-Low
	ENDIF
	;Calibrate High - From TrackView
	IF (D[995] = n) AND (D[996] = 12) AND (D[997] > 0) THEN
		NewHigh = StnRaw[n]
		IF (NewHigh > 0) AND (NewHigh < $FFFF) AND (NewHigh > StnLow) THEN
			D[4500 + n] = NewHigh
			D[4600 + n] = D[997]		;Test-Weight
		ENDIF
		D[996] = 0 ;Cancel the Cal-High
	ENDIF

	;Weigh Calculation - Multiply up to give accurate results
	HighLow = StnHigh - StnLow
	HighLow = HighLow * 1000
	;Avoid "Divide By Zero"
	IF (StnTestWgt > 0) THEN
		WeightUnits = DINT(HighLow / StnTestWgt)
		RawLow = INT(StnRaw[n] - StnLow)
		RawLow = RawLow * 1000
		IF (WeightUnits > 0) THEN ;AND (RawLow > 0) THEN
			Stn[n].Weight = INT(RawLow / WeightUnits)
		ELSE
			Stn[n].Weight = 0
		ENDIF
	ELSE
		Stn[n].Weight = 999
	ENDIF

	;Calibration Values to TrackView when requested equals current station
	IF (D32[230] = n) THEN
		D32[231] = UDINT(n)
		D32[232] = UDINT(StnLow)
		D32[233] = UDINT(StnHigh)
		D32[234] = UDINT(StnTestWgt)
		D32[235] = UDINT(StnRaw[n])
		D32[236] = UDINT(Stn[n].Weight)
	ENDIF

ENDLOOP

IF weighttest THEN
Stn[1].Weight = test1
Stn[2].Weight = test2
Stn[3].Weight = test3
Stn[4].Weight = test4
Stn[5].Weight = test4
Stn[6].Weight = test4
Stn[7].Weight = test4
Stn[8].Weight = test4
Stn[9].Weight = test4
Stn[10].Weight = test4
Stn[12].Weight = test1
Stn[11].Weight = test2
Stn[13].Weight = test3
Stn[14].Weight = test4
ENDIF
;Bag[101].Wgt = Stn[1].Weight
;Bag[102].Wgt = Stn[2].Weight
END_PROGRAM
```

### Program Logical/Sequences/zzAI2744 (IEC) - Weight 

#### zzAI2744Cyclic.ab - Cyclic code
```automation-basic
(********************************************************************
 * COPYRIGHT -- Kannegiesser UK Ltd
 ********************************************************************
 * Program: zzAI2744
 * File: zzAI2744Cyclic.ab
 * Author: zmclaren
 * Created: May 25, 2012
 ********************************************************************
 * Implementation of program zzAI2744
 ********************************************************************)

PROGRAM _CYCLIC
(* First we need to see if the last value is different to the previous one, *)
(* Then we will set the counters for each to zero *)
(* Also the Config Outputs will need setting to 0*)
IF (D[998] = 0) THEN
	LOOP i = 1 TO Std.MaxWeighstations DO
		myWeight = ((WeightRaw[i].Wgt_Channel_1 + WeightRaw[i].Wgt_Channel_2)/2)

		IF (LastRawValue[i] = myWeight)THEN        (* We have no change between the  two values *)
			IF (NoChangeCounter[i] >= 21) THEN          (* We need to reset the output back to zero *)
				WeightRaw[i].Config_Channel_1 = 0
				WeightRaw[i].Config_Channel_2 = 0
			ELSE
				IF (NoChangeCounter[i] = 20) THEN  (* We have had 20 cycles with no change on the input *)
					NoChangeCounter[i] = NoChangeCounter[i] + 1
					WeightRaw[i].Config_Channel_1  = %00110001  (* Make a change to both the Data Rate and the Range *)
					WeightRaw[i].Config_Channel_2  = %00110001
				ELSE
					NoChangeCounter[i] = NoChangeCounter[i] + 1  (* Increment the no change counter *)
				ENDIF
			ENDIF
		ELSE     (* There has been a change between the two  Values so store the old value and clear the counter *)
			LastRawValue[i] = myWeight (* Store the Last Value *)
			NoChangeCounter[i] = 0         (* Reset the Counter *)
			WeightRaw[i].Config_Channel_1 = 0      (* Leave the configuration as  0 *)
			WeightRaw[i].Config_Channel_2 = 0
		ENDIF
	ENDLOOP
ENDIF

END_PROGRAM
```

#### zzAI2744.var - Local variables
```iecst
(********************************************************************
 * COPYRIGHT -- Kannegiesser UK Ltd
 ********************************************************************
 * Program: zzAI2744
 * File: zzAI2744.var
 * Author: zmclaren
 * Created: May 25, 2012
 ********************************************************************
 * Local variables of program zzAI2744
 ********************************************************************)
VAR
	LastRawValue : ARRAY[0..199] OF DINT;
	i : UINT;
	NoChangeCounter : ARRAY[0..199] OF UINT;
	myWeight : DINT;
END_VAR
```

### Program Logical/Sequences/zzUld_4 (IEC)

#### zzuld_4.var
```iecst
VAR
	AutoRecirculation : BOOL;
END_VAR
VAR RETAIN
	AutoRepeat : BOOL;
	BagsRemaining : INT;
	BatchSize : UINT;
	BufferLineNum : ARRAY[0..19] OF UINT;
	PrgValid : BOOL;
	CurrentBag : UINT;
	CurrentDepth : UINT;
	CurrentLine : UINT;
	CustomerMode : UINT;
	CusValid : BOOL;
	DepthValid : BOOL;
	DepthValid2 : BOOL;
	Dest : UINT;
	Discharger : UINT;
	DischargerReady : BOOL;
	DischargerSpaces : INT;
	EndDischarger : UINT;
	EndLineSearch : UINT;
	ExpressBag : UINT;
	ExpressLine : UINT;
	FindBest : UINT;
	FoundBag : ARRAY[0..4] OF UINT;
	FoundLine : UINT;
	LastDischarger : UINT;
	LineDepthAllowed : ARRAY[0..49] OF USINT;
	LinesSearched : UINT;
	LineValid : BOOL;
	ManualBags : UINT;
	ManualBagsRecirc : UINT;
	ManualLine : UINT;
	ManualLineRecirc : UINT;
	MatchPrg1 : BOOL;
	MatchPrg2 : BOOL;
	MatchPrg3 : BOOL;
	MixCustomers : BOOL;
	n : UINT;
	NoBagAvailable : BOOL;
	PLS : BOOL;
	PriorityLine : UINT;
	ProgQtyComplete : UINT;
	ProgramFinished : BOOL;
	ProgramReset : BOOL;
	ProgramRunning : BOOL;
	ProgramStep : UINT;
	Quantity : UINT;
	RecircDest : UINT;
	RecircSpaces : INT;
	RecircSpacesRemain : UINT;
	RecirculationMaxDepth : UINT;
	RegOffset : ARRAY[0..19] OF UINT;
	ScanCount : UINT;
	SearchPrg : ARRAY[0..3] OF UINT;
	SearchCus : ARRAY[0..3] OF UDINT;
	SearchLine : UINT;
	SearchSpaces : UINT;
	SkipIncompleteStep : BOOL;
	SpacesUsed : UINT;
	StartDischarger : UINT;
	StartLine : UINT;
	StartLineSearch : UINT;
	StepsSearched : UINT;
	TestDischarger : UINT;
	UldStep : UINT;
END_VAR
VAR
	UnloadingMaxDepth : UINT;
END_VAR
VAR RETAIN
	UnusedStep : BOOL;
	x : UINT;
	MixPrograms : BOOL;
END_VAR
VAR
	CatValid : BOOL;
	BagsWithDest : UINT;
	DstValid : BOOL;
	RecircLimit : INT;
	SkipLineStart : UINT;
	SkipLineEnd : UINT;
	LineValid2 : BOOL;
	BagValid : BOOL;
	DischLimit : UINT;
	StartStopOffset : UINT;
	LineValid3 : BOOL;
	TimTest : UINT;
	TestPLS : BOOL;
	RecircBag : UINT;
END_VAR
```

#### zzuld_4.ab
```automation-basic
;Unloading Programs 4 - Search and give Destination (Using Bag)

	;-----------------------------------------------------------
	;Version 1.00 03/12/2005 D.J. First Issue
	;Version 2.00 30/08/2007 D.J. BagRemaining changed to INT
	;Version 3.00 25/06/2009 D.J. Use .Prg Instead of .Cat
	;Version 4.00 09/11/2009 D.J. Allow multiple destination
	;Version 4.10 08/06/2011 D.J. Addes Start/Stop for each line
	;-----------------------------------------------------------

PROGRAM _INIT

	;Constants
	;---------

	UnloadingMaxDepth 	= 1 ;Set with Batch Size and Scan Time in mind 8 = Standard MAX BAG AMT CALL OFF

	StartDischarger 	= 1
	EndDischarger   	= 2 ;Allowed for 3rd future discharger so recirc takes dest 24

	StartLineSearch 	= 1
	EndLineSearch 		= 7 ;Include Lines A-C

	SkipLineStart		= 0
	SkipLineEnd			= 0

	RegOffset[1]    	= 1000
	RegOffset[2]    	= 1200
	RegOffset[3]    	= 1400
	RegOffset[4]    	= 1600
	RegOffset[5]    	= 1800
	RegOffset[6]    	= 2000
	RegOffset[7]    	= 2200
	RegOffset[8]    	= 2400

	;Enter Line Number for Discharger buffers - Recirc is after last Discharger
	;Destination Code bag will be allocated
	BufferLineNum[1]	= 11
	BufferLineNum[2]	= 12
	BufferLineNum[3]	= 13
	BufferLineNum[4]	= 14
	BufferLineNum[5]	= 15
	BufferLineNum[6]	= 16
	BufferLineNum[7]	= 17
	BufferLineNum[8]	= 18

	RecircDest			= 10

	PriorityLine		= 0		;Always Search this line first then use the Uld[n].DischargerStartLine Set to 0 if not required

	StartStopOffset		= 40;200	;Offset for D register for each lines Start / Stop ie D201 to D2xx - Set to Zero if no Start / Stops

END_PROGRAM

PROGRAM _CYCLIC

	;Spare Step
	IF (UldStep = 0) THEN
		UldStep = 1
	ENDIF

	;UldStep 1	- Check no bags in Storage are allocated with a destination
	IF (UldStep = 1) THEN

		;Set ScanCount as alternating Value 25 is about 5 seconds
		IF (ScanCount = 1) THEN
			Discharger 	= (Discharger + 1)
			ScanCount 	= 0
		ENDIF

		ScanCount = (ScanCount + 1)

		IF ((Discharger > EndDischarger) OR (Discharger < StartDischarger))  THEN
			Discharger 	= StartDischarger
		ENDIF

		;Set discharger number in TestDischarger if required
		IF (TestDischarger > 0) THEN
			Discharger = TestDischarger
		ENDIF

		;Read Program Variables
		n = RegOffset[Discharger]

		ProgramStep 			= D[1 + n]
		ProgQtyComplete			= D[2 + n]
		AutoRecirculation 		= (D[1003] = 1)		;Use if Re-cirulation or Offgoing Batching Loop
		RecirculationMaxDepth 	= D[1004]

		ManualLine       		= D[7 + n]
		ManualBags       		= D[8 + n]
		StepsSearched			= D[9 + n]
		SkipIncompleteStep 		= (D[10 + n] = 1)
		AutoRepeat				= (D[11 + n] = 1)
		MixPrograms 			= (D[12 + n] = 1)	;Batch must be same Program?
		MixCustomers 			= (D[13 + n] = 1) 	;Batch must be same Customer?
		NoBagAvailable			= (D[14 + n] = 1)	;Alarm 'No Bag Available'
		ProgramFinished			= (D[15 + n] = 1)	;Alarm 'Finished Program'
		ManualLineRecirc 		= D[1016]
		ManualBagsRecirc 		= D[1017]
		ProgramRunning			= (D[19 + n] = 1)	;Run from TrackView
		ExpressLine 			= D[20 + n]
		CustomerMode			= D[21 + n]			;Customer Mode 0 = Normal Manual, 1 = Reset Pointer on every step, 2 = Check all steps before changing
		ProgramReset			= (D[22 + n] = 1)	;Customer FIFO Reset

		DischargerReady			= Uld[Discharger].SDCReady

		DischargerSpaces 		= Line[BufferLineNum[Discharger]].SpaceBIT

		;Calculate RecircSpaces
		RecircSpaces  		= (DestCountSystem[RecircDest] - DestCountStorage[RecircDest])
		IF (RecircSpaces < 0) THEN ; Keep value positive
			RecircSpaces = 0
		ENDIF
		BagsWithDest 			= DestCountStorage[BufferLineNum[Discharger]]

		IF ((BagsWithDest = 0) AND (Discharger > 0)) THEN
			UldStep = 2
		ELSE
			;Allow program to skip blank steps when Bags Have Destinations
			UnusedStep		= (D[40 + n + ProgramStep] = 0) ;Bags = 0
			IF UnusedStep THEN
				UldStep = 15
			ENDIF
		ENDIF

		;If program is new then Clear Search Values
		IF ProgramReset THEN
			Uld[Discharger].FIFOCustomer 		= 0	;Clear Current Customer - FIFO Will allocate next
			Uld[Discharger].LastCustQtyComplete = 0	;Clear Last Quantity
			StepsSearched 						= 0	;Clear Steps Searched / Failed
			D[22 + n]	 						= 0 ;Clear Program Reset
			UldStep 							= 0	;Keep Unloading Step at 0 to allow Customer FIFO to allocate next Customer
		ENDIF

	ENDIF

	;UldStep 2	- Check for a Manual Re-circulation regardless of Discharger
	;			- Note will stop all unloading progrms if not ready
	IF (UldStep = 2) THEN
		IF ((ManualLineRecirc >= StartLineSearch) AND (ManualLineRecirc <= EndLineSearch) AND (ManualBagsRecirc > 0)) THEN
			IF Uld[EndDischarger + 1].SDCReady THEN
				UldStep = 21
			ELSE
				UldStep = 0
			ENDIF
		ELSE
			UldStep = 3
		ENDIF
	ENDIF

	;UldStep 3	- Check Discharger is Ready
	IF (UldStep = 3) THEN
		IF (DischargerReady AND ProgramRunning) THEN; AND (DischargerSpaces > 0)) THEN
			UldStep = 4
		ELSE
			;If not ready then clear steps searched
			UldStep = 0
		ENDIF
	ENDIF

	;UldStep 4	- Check for a Manual Bags
	IF (UldStep = 4) THEN
		IF ((ManualLine >= StartLineSearch) AND (ManualLine <= EndLineSearch) AND (ManualBags > 0)) THEN
			UldStep = 22
		ELSE
			UldStep = 5
		ENDIF
	ENDIF

	;STEP 5	- Check Express Line
	IF (UldStep = 5) THEN
		IF (ExpressLine > 0) THEN
			ExpressBag  = Line[ExpressLine].FirstBag
		ENDIF
		IF ((Bag[ExpressBag].Cat > 0) AND (ExpressLine > 0) AND (Line[BufferLineNum[Discharger]].SpaceBIT > 0)) THEN
			UldStep = 23
		ELSE
			UldStep = 6
		ENDIF
	ENDIF

	;UldStep 6	- Check Program step
	IF (UldStep = 6) THEN

		;Check if UldStep Valid
		IF (ProgramStep < 1) OR (ProgramStep > 20) THEN
			ProgramStep = 1 					;Set to UldStep 1
			ProgQtyComplete = 0 				;Clear Qty Completed
			IF (CustomerMode = 1) THEN
				Uld[Discharger].FIFOCustomer = 0
			ENDIF
		ENDIF

		UldStep = 7

	ENDIF

	;UldStep 7 - Check for remaining bags on the current Step
	IF (UldStep = 7) THEN

		BatchSize 		= D[80 + n + ProgramStep]
		Quantity 		= D[40 + n + ProgramStep] ;* BatchSize ;Take bags * BatchSize
		BagsRemaining 	= INT(Quantity - ProgQtyComplete)

		IF ((BagsRemaining > 0) AND (BagsRemaining >= INT(BatchSize))) THEN
			UldStep = 8
		ELSE
			UldStep = 15 ;Step Not Complete Or No Qty
		ENDIF

	ENDIF

	;UldStep 8 - Check the 'Batch' Will fit onto the Buffer
	IF (UldStep = 8) THEN

		BatchSize 		= D[80 + n + ProgramStep]

		IF (DischargerSpaces >= BatchSize) THEN
			UldStep = 9
		ELSE
			UldStep = 0
		ENDIF

	ENDIF

	;UldStep 9 - Set Search Values
	IF (UldStep = 9) THEN

		IF (PriorityLine = 0) THEN
			StartLine = (Uld[Discharger].DischargerStartLine + 1)
			IF ((StartLine < StartLineSearch) OR (StartLine > EndLineSearch)) THEN
				StartLine = StartLineSearch
			ENDIF
		ELSE
			StartLine = PriorityLine
		ENDIF

		SearchLine   = D[60 + n + ProgramStep]
		BatchSize    = D[80 + n + ProgramStep]

		SearchPrg[1] = D[100 + n + ProgramStep]
		SearchPrg[2] = D[120 + n + ProgramStep]
		SearchPrg[3] = D[140 + n + ProgramStep]

		IF (CustomerMode = 0) THEN
			SearchCus[1] = D32[20 + Discharger]					;Manually Selected Customer
		ELSE
			SearchCus[1] = Uld[Discharger].FIFOCustomer ;Automatic FIFO Customer Selection
		ENDIF

		SearchSpaces = 0 ;Search Always starts with no spaces on the recirc

		UldStep = 10

	ENDIF

	;UldStep 10 - Search for Bag(s) could be modified to run over several scans to reduce its load on the PLC
	;			  To find the best pos using set RecircSpaces low increasing to max.
	IF (UldStep = 10) THEN

		LOOP FindBest = 1 TO 3 DO

			;Clear the Search Array and Set Depth Allowed 1 for upto 49 storage lines
			FoundLine = 0
			memset(ADR(FoundBag[0]),0,10)
			memset(ADR(LineDepthAllowed[0]),1,50)

			RecircSpacesRemain = SearchSpaces

			;Can the 1st, 2nd or 3rd Program be mixed with each other? 'Mix Programs'
			IF (FindBest = 1) THEN
				MatchPrg1 = TRUE
				MatchPrg2 = FALSE
				MatchPrg3 = FALSE
			ELSE IF (FindBest = 2) THEN
				MatchPrg1 = MixPrograms
				MatchPrg2 = TRUE
				MatchPrg3 = FALSE
			ELSE
				MatchPrg1 = MixPrograms
				MatchPrg2 = MixPrograms
				MatchPrg3 = TRUE
			ENDIF

			;Loop around all the storage lins row by row.
			LOOP CurrentDepth = 1 TO UnloadingMaxDepth DO ;Always search to max depth to check scan time

				;CurrentLine = StartLine

				LOOP LinesSearched = StartLineSearch TO EndLineSearch DO ;Loop around each line

					CurrentLine = LongestTime[LinesSearched]
					CurrentBag = (Line[CurrentLine].FirstBag + (CurrentDepth - 1))

					;Search / Add
					;------------
					;For Unloading by line - If there is a bag on the line and the 1st Program = 0 then check Customer valid
					;eg if the 1st Prg and 1st Cus are set to 0 then this would set "CatCusValid" to TRUE but the line must also match
					;Unloading by Customer only cannot be done.

					CatValid = (Bag[CurrentBag].Cat > 0)
					CusValid = FALSE
					PrgValid = FALSE
					DstValid = FALSE

					;Check the Destination is valid (allow dischargers to take recirc bags)
					IF ((Bag[CurrentBag].Dst = 0) OR (Bag[CurrentBag].Dst = RecircDest)) THEN
						DstValid = TRUE
					ENDIF

					;Check the Customer is valid
					IF (Bag[CurrentBag].Cus = SearchCus[1]) THEN
						CusValid = TRUE
					ELSE IF ((SearchCus[1] = 0) AND (CustomerMode = 0)) THEN ;Only Valid If Manual Customer Selection
						CusValid = TRUE
					ENDIF

					;Check the Category is valid
					IF (MatchPrg1 AND (Bag[CurrentBag].Prg = SearchPrg[1]) AND (SearchPrg[1] > 0)) THEN
						PrgValid = TRUE
					ENDIF
					IF (MatchPrg2 AND (Bag[CurrentBag].Prg = SearchPrg[2]) AND (SearchPrg[2] > 0)) THEN
						PrgValid = TRUE
					ENDIF
					IF (MatchPrg3 AND (Bag[CurrentBag].Prg = SearchPrg[3]) AND (SearchPrg[3] > 0)) THEN
						PrgValid = TRUE
					ENDIF
					;If Unloading by line and no Category is set then Set Valid
					IF ((Bag[CurrentBag].Cat > 0) AND (SearchPrg[1] = 0) AND (SearchLine > 0)) THEN
						PrgValid = TRUE
					ENDIF

					BagValid = (CurrentBag >= Line[CurrentLine].FirstBag) AND (CurrentBag <= Line[CurrentLine].LastBag)

					LineValid 	= ((SearchLine = CurrentLine) OR (SearchLine = 0))
					LineValid2 	= ((CurrentLine < SkipLineStart) OR (CurrentLine > SkipLineEnd))
					IF (StartStopOffset < 100) THEN
						LineValid3	= ((StartStopOffset = 0) OR (D[StartStopOffset + CurrentLine] > 0))
					ELSE
						LineValid3	= (D[StartStopOffset + 7600 + CurrentLine] > 0) ;Start / Stop 100 -299 D7700 to D7899
					ENDIF

					DepthValid	= ((LineDepthAllowed[CurrentLine] + RecircSpacesRemain) >= CurrentDepth)
					DepthValid2	= ((CurrentDepth <= RecirculationMaxDepth) OR NOT AutoRecirculation)

					IF (BagValid AND DstValid AND CatValid AND PrgValid AND CusValid AND LineValid AND LineValid2 AND LineValid3 AND DepthValid AND DepthValid2) THEN

						IF (FoundBag[0] < BatchSize)  THEN
							FoundBag[0] = FoundBag[0] + 1
							x 			= FoundBag[0]
							FoundBag[x] = CurrentBag
							FoundLine	= CurrentLine

							;If bags need to go to recirc then dec
							IF (LineDepthAllowed[CurrentLine] < USINT(CurrentDepth)) THEN
								SpacesUsed 			= USINT(CurrentDepth) - LineDepthAllowed[CurrentLine]
								RecircSpacesRemain 	= (RecircSpacesRemain - SpacesUsed)
							ENDIF

							LineDepthAllowed[CurrentLine] = USINT(CurrentDepth + 1)

						ENDIF

					ENDIF

					;-------------
					;End of Search
					;-------------

					;If searching using priority line then start from the Discharger Start Line
					IF CurrentLine = PriorityLine THEN
						CurrentLine = (Uld[Discharger].DischargerStartLine)
					ENDIF

					;Set Next Line
					CurrentLine = (CurrentLine + 1)
					IF CurrentLine > EndLineSearch THEN
						CurrentLine = StartLineSearch
					ENDIF

					;If the new line = priority line then skip as its already been searched
					IF CurrentLine = PriorityLine THEN
						CurrentLine = (CurrentLine + 1)
						IF CurrentLine > EndLineSearch THEN
							CurrentLine = StartLineSearch
						ENDIF
					ENDIF

				ENDLOOP

			ENDLOOP

			EXITIF FoundBag[0] = BatchSize

		ENDLOOP				;Find Best

		;Check if the bags were found
		IF FoundBag[0] = BatchSize THEN
			UldStep = 14 	;Action Results
		ELSE IF (AutoRecirculation AND (RecircSpaces > SearchSpaces) AND (RecircSpaces > 0)) THEN
			;If recirculation - to find the best possible result inc the search spaces each scan
			;until total spaces searched
			SearchSpaces = (SearchSpaces + 1)
			UldStep = 10	;Try with more recirculation space
		ELSE
			UldStep = 15	;Search Failed
		ENDIF

	ENDIF

	;UldStep 14 - Search Valid give bags destinations, inc qty taken by batchsize
	IF (UldStep = 14) THEN

		LOOP Dest = 1 TO BatchSize DO
			Bag[FoundBag[Dest]].Dst = USINT(BufferLineNum[Discharger])
		ENDLOOP
		ProgQtyComplete = ProgQtyComplete + BatchSize	;Inc Qty Completed
		StepsSearched = 0 								;Clear the search failed UldStep counter
		NoBagAvailable = FALSE 							;No Bags Alarm (OFF)
		LastDischarger = Discharger

		IF AutoRecirculation THEN
			UldStep = 24		;Set Any Bags for Auto-Reirculation
		ELSE
			UldStep = 0
		ENDIF

		;Mode 2 Needs to keep the Qty completed for the next customer
		Uld[Discharger].LastCustQtyComplete = ProgQtyComplete

	ENDIF

	;UldStep 15 - Search Failed
	IF (UldStep = 15) THEN

		BatchSize 		= D[80 + n + ProgramStep]
		;Quantity 		= D[40 + n + ProgramStep] * BatchSize ;Take bags * BatchSize
		Quantity		= (D[40 + n + ProgramStep])
		BagsRemaining 	= INT(Quantity - ProgQtyComplete)
		UnusedStep		= (D[40 + n + ProgramStep] = 0) ;Bags = 0

		;Inc Steps searched counter
		IF (StepsSearched < 21) THEN
			StepsSearched = (StepsSearched + 1)
		ENDIF

		IF (CustomerMode = 0) THEN
			IF (BagsRemaining <= 0) THEN
				UldStep = 16			;Try Next Step
			ELSE IF (SkipIncompleteStep OR UnusedStep) THEN
				UldStep = 16			;Try Next Step
			ELSE
				NoBagAvailable = TRUE 	;Set Alarm and Wait for Operator to change Program or More Bags
				UldStep = 0
			ENDIF
		ENDIF

		IF (CustomerMode = 1) THEN
			IF (BagsRemaining <= 0) THEN
				UldStep = 16			;Try Next Step
			ELSE IF (NOT UnusedStep) THEN
				IF (Uld[Discharger].FIFONextCustomer > 0) THEN
					;Mode 1 Search again with the Next Customer Without Changing Step
					Uld[Discharger].FIFOCustomer = Uld[Discharger].FIFONextCustomer
					UldStep = 0
				ELSE
					;Last customer was not found reset FIFO position to 1 and keep searching
					Uld[Discharger].FIFOCustomer = 0 ;Reset the First Customer
					NoBagAvailable = TRUE
					UldStep = 0
				ENDIF
			ELSE IF (SkipIncompleteStep OR UnusedStep) THEN
				UldStep = 16			;Try Next Step
			ELSE
				NoBagAvailable = TRUE	;Set Alarm and Wait for Operator to change Program or More Bags
				UldStep = 0
			ENDIf
		ENDIF

		IF (CustomerMode = 2) THEN
			IF (BagsRemaining <= 0) THEN
				UldStep = 16			;Try Next Step
			ELSE IF (StepsSearched = 21) THEN
				IF (Uld[Discharger].FIFONextCustomer > 0) THEN
					;Mode 2 Customer Change Only After 21 Steps Searched
					Uld[Discharger].FIFOCustomer = Uld[Discharger].FIFONextCustomer
					ProgQtyComplete = Uld[Discharger].LastCustQtyComplete
					StepsSearched = 0 ;FREI Use -1 to go to next step
					UldStep = 0
				ELSE
					;Last customer was not found reset FIFO position to 1 and keep searching
					Uld[Discharger].FIFOCustomer = 0 ;Reset the First Customer
					NoBagAvailable = TRUE
					StepsSearched = 0
					UldStep = 0
				ENDIF
			ELSE IF (SkipIncompleteStep OR UnusedStep) THEN
				UldStep = 16			;Try Next Step
			ELSE
				NoBagAvailable = TRUE	;Set Alarm and Wait for Operator to change Program or More Bags
				UldStep = 0
			ENDIF
		ENDIF

	ENDIF

	;Skip Program Step or Set to 1
	IF (UldStep = 16) THEN
		IF (ProgramStep = 20) THEN
			IF AutoRepeat THEN
				ProgramStep = 1
				IF (CustomerMode = 1) THEN
					Uld[Discharger].FIFOCustomer = 0 ;Start Search With First Customer
				ENDIF
			ELSE
				ProgramFinished = TRUE
			ENDIF
		ELSE
			ProgramStep = ProgramStep + 1
			IF (CustomerMode = 1) THEN
				Uld[Discharger].FIFOCustomer = 0 ;Start Search With First Customer
			ENDIF
		ENDIF
		ProgQtyComplete = 0
		UldStep = 0
	ENDIF

	;UldStep 21 -	Manual Bags Recirc
	IF (UldStep = 21) THEN

		LOOP RecircBag = 0 TO (ManualBagsRecirc - 1) DO

			CurrentBag = (Line[ManualLineRecirc].FirstBag + RecircBag)

			IF Bag[CurrentBag].Cat > 0 THEN
				Bag[CurrentBag].Dst = USINT(RecircDest)	;Set Destination
				;ManualBagsRecirc    = (ManualBagsRecirc - 1)					;Dec manual bags by 1
			ENDIF
		ENDLOOP
		ManualBagsRecirc = 0
		UldStep = 0

	ENDIF

	;UldStep 22 - Manual Bags to Discharger
	IF (UldStep = 22) THEN

		CurrentBag = Line[ManualLine].FirstBag

		IF Bag[CurrentBag].Cat > 0 THEN
			Bag[CurrentBag].Dst = USINT(BufferLineNum[Discharger])
			ManualBags 			= (ManualBags - 1)				;Dec manual bags by 1
		ENDIF

		UldStep = 0

	ENDIF

	;UldStep 23 - Express Line
	IF (UldStep = 23) THEN

		Bag[ExpressBag].Dst = USINT(BufferLineNum[Discharger])

		UldStep = 0

	ENDIF

	;UldStep 24 - Set Bags to re-circulation line if they need to move out of the way of bags with destinations
	IF (UldStep = 24) THEN

		LOOP CurrentLine = StartLineSearch to EndLineSearch DO
			LOOP CurrentBag = Line[CurrentLine].LastBag DOWNTO Line[CurrentLine].FirstBag DO

				IF (Bag[CurrentBag].Dst > 0) AND (Bag[CurrentBag - 1].Dst = 0) AND (CurrentBag > Line[CurrentLine].FirstBag) THEN
					Bag[CurrentBag - 1].Dst = USINT(RecircDest)
				ENDIF

			ENDLOOP
		ENDLOOP

		UldStep = 0

	ENDIF

	;Outputs
	;-------

	D[1 + n] 		= ProgramStep
	D[2 + n]		= ProgQtyComplete
	D[8 + n] 		= ManualBags
	D[9 + n]		= StepsSearched

	;No bag available is displayed if 20 steps have been searched and program is running
	IF (NoBagAvailable AND ProgramRunning) THEN
		D[14 + n] = 1
		Alarm[Discharger + 200].On		= TRUE
		Alarm[Discharger + 200].Bag 	= 0
		Alarm[Discharger + 200].Name 	= almUldNoBag
		Alarm[Discharger + 200].Beacon	= FALSE
	ELSE
		D[14 + n]	= 0
	ENDIF

	;Program is only finished if on step 20 and Program Running
	IF (ProgramFinished AND ProgramRunning AND (ProgramStep = 20)) THEN
		D[15 + n]	= 1
		Alarm[Discharger + 200].On		= TRUE
		Alarm[Discharger + 200].Bag 	= 0
		Alarm[Discharger + 200].Name 	= almUldProgFinished
		Alarm[Discharger + 200].Beacon	= FALSE
	ELSE
		D[15 + n]	= 0
	ENDIF

	;If no unloading alarms then clear unloading alarm
	IF (D[14 + n] = 0) AND (D[15 + n] = 0) THEN
		Alarm[Discharger + 200].On		= FALSE
		Alarm[Discharger + 200].Bag 	= 0
		Alarm[Discharger + 200].Name 	= almNoAlarm
		Alarm[Discharger + 200].Beacon	= FALSE
	ENDIF

	D[1017]		= ManualBagsRecirc

	IF ProgramRunning THEN
		D[18 + n]	= 1
	ELSE
		D[18 + n]	= 0
	ENDIF

	D32[30 + Discharger] 	= Uld[Discharger].FIFOCustomer
	;D[187 + n] 		= Uld[Discharger].FIFONextCustomer

END_PROGRAM
```

### Program Logical/Sequences/zzGetNames (IEC)

#### zzGetNames.var
```iecst
(********************************************************************
 * COPYRIGHT --
 ********************************************************************
 * Program: zzGetNames
 * File: zzGetNames.var
 * Author: Dave
 * Created: November 19, 2010
 ********************************************************************
 * Local variables of program zzGetNames
 ********************************************************************)
VAR
	MaxDisplays : UINT;
	OwnerID : UDINT;
	TviewReplyOwnerID : UDINT;
	WaitReply : BOOL;
	myBag : UINT;
	CommsID : UDINT;
	Timer2Q : BOOL;
	Timer1Q : BOOL;
	Timer1ET : UDINT;
	Timer2ET : UDINT;
END_VAR
```

#### zzGetNames.ab
```automation-basic
(********************************************************************
 * COPYRIGHT --
 ********************************************************************
 * Program: zzGetNames
 * File: zzGetNames.ab
 * Author: Dave
 * Created: November 19, 2010
 ********************************************************************
 * Implementation of program zzGetNames
 ********************************************************************)

;Get names from TrackView - Program, Category and Customer

;Version 1.00 19/11/2010 D.J. First Issue
;Version 2.00 12/12/2010 D.J. Added default values
;Version 3.00 19/10/2011 D.J. Clear Name when number has changed - if no TrackView then name will remain clear.

;Enter the required bag numbers for collection of names. Use the resulting names in transmisions to displays.

PROGRAM _INIT

	zzGetNamesData[1].BagNumber = 101
	zzGetNamesData[2].BagNumber = 102
	zzGetNamesData[3].BagNumber = 103
	zzGetNamesData[4].BagNumber = 104
	zzGetNamesData[5].BagNumber = 0
	zzGetNamesData[6].BagNumber = 0
	zzGetNamesData[7].BagNumber = 0
	zzGetNamesData[8].BagNumber = 0
	zzGetNamesData[9].BagNumber = 0
	zzGetNamesData[10].BagNumber = 0
	zzGetNamesData[11].BagNumber = 0
	zzGetNamesData[12].BagNumber = 0
	zzGetNamesData[13].BagNumber = 0
	zzGetNamesData[14].BagNumber = 0
	zzGetNamesData[15].BagNumber = 0
	zzGetNamesData[16].BagNumber = 0

	MaxDisplays = 16
	IF (MaxDisplays > SIZEOF(zzGetNamesData)) THEN
		MaxDisplays = SIZEOF(zzGetNamesData)
	ENDIF

	WaitReply = FALSE

	zzGetNamesData[0].BagNumber = 1
	zzGetNamesData[0].Prg		= 1
	strcpy(ADR(zzGetNamesData[0].PrgLong),"PRG")
	strcpy(ADR(zzGetNamesData[0].PrgName),"ProgramName")
	zzGetNamesData[0].Cat		= 1
	strcpy(ADR(zzGetNamesData[0].CatLong),"CAT")
	strcpy(ADR(zzGetNamesData[0].CatName),"CategoryName")
	zzGetNamesData[0].Cus		= 1
	strcpy(ADR(zzGetNamesData[0].CusLong),"CUS")
	strcpy(ADR(zzGetNamesData[0].CusName),"CustomerName")

END_PROGRAM

PROGRAM _CYCLIC

	;Search for display data that needs updating
	IF NOT WaitReply THEN

		OwnerID = OwnerID + 1
		IF (OwnerID > MaxDisplays) THEN
			OwnerID = 1
		ENDIF

		myBag = zzGetNamesData[OwnerID].BagNumber

		IF ((zzGetNamesData[OwnerID].Prg <> Bag[myBag].Prg) AND (Bag[myBag].Prg > 0)) THEN
			memcpy(ADR(zzGetNamesData[OwnerID].PrgLong),ADR(""),8)
			memcpy(ADR(zzGetNamesData[OwnerID].PrgName),ADR(""),32)
			WaitReply = TRUE
		ENDIF

		IF ((zzGetNamesData[OwnerID].Cat <> Bag[myBag].Cat) AND (Bag[myBag].Cat > 0)) THEN
			memcpy(ADR(zzGetNamesData[OwnerID].CatLong),ADR(""),8)
			memcpy(ADR(zzGetNamesData[OwnerID].CatName),ADR(""),32)
			WaitReply = TRUE
		ENDIF

		IF ((zzGetNamesData[OwnerID].Cus <> Bag[myBag].Cus) AND (Bag[myBag].Cus > 0)) THEN
			memcpy(ADR(zzGetNamesData[OwnerID].CusLong),ADR(""),8)
			memcpy(ADR(zzGetNamesData[OwnerID].CusName),ADR(""),32)
			WaitReply = TRUE
		ENDIF

		;Set TrackView Registers
		IF WaitReply THEN
			CommsID = CommsID + 1
			IF (CommsID > $7FFFFFFF) THEN
				CommsID = 1
			ENDIF
			D32[201] = OwnerID
			D32[202] = CommsID
			D32[204] = UDINT(Bag[myBag].Prg)
			D32[205] = Bag[myBag].Cat
			D32[206] = Bag[myBag].Cus
		ENDIF

	ENDIF

	TviewReplyOwnerID = D32[203]

	;Set request to TrackView until reply
	IF (WaitReply AND (CommsID = TviewReplyOwnerID)) THEN

		myBag = zzGetNamesData[OwnerID].BagNumber

		zzGetNamesData[OwnerID].Prg = Bag[myBag].Prg
		memcpy(ADR(zzGetNamesData[OwnerID].PrgLong),ADR(D32[531]),8)
		memcpy(ADR(zzGetNamesData[OwnerID].PrgName),ADR(D32[533]),32)

		zzGetNamesData[OwnerID].Cat = Bag[myBag].Cat
		memcpy(ADR(zzGetNamesData[OwnerID].CatLong),ADR(D32[541]),8)
		memcpy(ADR(zzGetNamesData[OwnerID].CatName),ADR(D32[543]),32)

		zzGetNamesData[OwnerID].Cus = Bag[myBag].Cus
		memcpy(ADR(zzGetNamesData[OwnerID].CusLong),ADR(D32[551]),8)
		memcpy(ADR(zzGetNamesData[OwnerID].CusName),ADR(D32[553]),32)

		WaitReply 	= FALSE

	ENDIF

END_PROGRAM
```

### Package Logical/Timestamp - Keeps current timestamp

### Program Logical/Timestamp/zzGetTime

#### zzGetTime.var
```iecst
(********************************************************************
 * COPYRIGHT -- HP
 ********************************************************************
 * Program: zzGetTime
 * File: zzGetTime.var
 * Author: treamsbottom
 * Created: June 04, 2014
 ********************************************************************
 * Local variables of program zzGetTime
 ********************************************************************)
VAR
	GetTimeStamp : DTGetTime;
	setTimeStamp : DTSetTime;
	enable : BOOL;
	DT1 : DATE_AND_TIME;
	status : UINT;
	kev : BOOL;
END_VAR
```

#### zzGetTimeCyclic.ab
```automation-basic
(********************************************************************
 * COPYRIGHT -- HP
 ********************************************************************
 * Program: zzGetTime
 * File: zzGetTimeCyclic.ab
 * Author: treamsbottom
 * Created: June 04, 2014
 ********************************************************************
 * Implementation of program zzGetTime
 ********************************************************************)

PROGRAM _CYCLIC
;enable = Std.Clock1s

;;DT1 = DT#2023-01-21-11:03                       (* actual time *)
;DTSetTime(enable,DT1,status)

	GetTimeStamp.enable = TRUE
	GetTimeStamp FUB DTGetTime()
	IF GetTimeStamp.status = ERR_OK THEN
		CurrentTimestamp = GetTimeStamp.DT1
	ENDIF
	D32[78] = UDINT(CurrentTimestamp);

;	//Set the current time.
	//DTSetTime(enable, DT1, status)
;	setTimeStamp.enable := (D32[78] > 0)
;	setTimeStamp.DT1 := DT(D32[78]); 	CAST D32 TO DT
;	setTimeStamp FUB DTSetTime()
;	IF (setTimeStamp.status =  ERR_OK) THEN
;		D32[79] = 0
;	ENDIF
;
END_PROGRAM
```

### Package Logical/Data_BackUp - *Handles all data back up

### Program Logical/Data_BackUp/zzDataStore (IEC) - *Store all data

#### zzDataStore.ab - Implementation code
```automation-basic
(********************************************************************
 * COPYRIGHT -- HP
 ********************************************************************
 * Program: zzDataStore
 * File: zzDataStore.ab
 * Author: treamsbottom
 * Created: March 20, 2014
 ********************************************************************
 * Implementation of program zzDataStore
 ********************************************************************)
;-- V1.01 21-03-2014 First Version-- TR.

PROGRAM _INIT
;Set Global Memtype
MemType = doSYSROM
pUSBDevice = ADR("USBStick")

;Set the Data to be backed up
;Name must be 10 chars max
Backup[0].MemTyp = MemType
Backup[0].DataLength = SIZEOF(Bag)
Backup[0].pData 	= ADR(Bag)
Backup[0].pFileName	= ADR("Bak_Bag")

Backup[1].MemTyp = MemType
Backup[1].DataLength = SIZEOF(C)
Backup[1].pData 	= ADR(C)
Backup[1].pFileName	= ADR("Bak_C")

Backup[2].MemTyp = MemType
Backup[2].DataLength = SIZEOF(D)
Backup[2].pData 	= ADR(D)
Backup[2].pFileName	= ADR("Bak_D")

Backup[3].MemTyp = MemType
Backup[3].DataLength = SIZEOF(D32)
Backup[3].pData 	= ADR(D32)
Backup[3].pFileName	= ADR("Bak_D32")

Backup[4].MemTyp = MemType
Backup[4].DataLength = SIZEOF(ReportBuffer)
Backup[4].pData 	= ADR(ReportBuffer)
Backup[4].pFileName	= ADR("Bak_Report")

Backup[5].MemTyp = MemType
Backup[5].DataLength = SIZEOF(RB_Posn)
Backup[5].pData 	= ADR(RB_Posn)
Backup[5].pFileName	= ADR("Bak_RBPosn")

Backup[6].MemTyp = MemType
Backup[6].DataLength = SIZEOF(RB_Perm)
Backup[6].pData 	= ADR(RB_Perm)
Backup[6].pFileName	= ADR("Bak_RBPerm")

Backup[7].MemTyp = MemType
Backup[7].DataLength = SIZEOF(SQL)
Backup[7].pData 	= ADR(SQL)
Backup[7].pFileName	= ADR("Bak_SQL")

;Backup[8].MemTyp = MemType
;Backup[8].DataLength = SIZEOF(RFIDCode)
;Backup[8].pData 	= ADR(RFIDCode)
;Backup[8].pFileName	= ADR("Bak_RFID")

MaxBackUpAreas = 7

END_PROGRAM

PROGRAM _CYCLIC
IF TestTIM THEN
	memcpy(ADR(D),1,100000)
	TestTIM = FALSE
ENDIF
myMonitorReg = 291 ; D reg to monitor if 0 then stop back up
myUpdateReg	= 292 ; Reply reg from Trackview used to restore data.
myAlarm = 209

Alarm[myAlarm].On	= FALSE
Alarm[myAlarm].Bag 	= 0
Alarm[myAlarm].Name	= 0

CASE eBackup OF
	ACTION eNull:
		IF (D[myUpdateReg] = cBackUp_FromSYSROM) THEN
			;Registers are updated when Read completes
			eBackup = eRead
		ELSE IF (D[myUpdateReg] = cBackUp_FromUSB) THEN
			D[myUpdateReg] = 0
			eBackup = eReadFromUSB
		ELSE IF (D[myUpdateReg] = cBackUp_StartWithoutRestore) THEN
			D[myMonitorReg] = 1
			D[myUpdateReg] = 0
		ELSE
			D[myUpdateReg] = 0
			 IF (D[myMonitorReg] > 0) THEN
				eBackup = eWrite
			ENDIF
		ENDIF
		n = 0
	ENDACTION

	ACTION eWrite: ; Back up perm memory
		BackUp.Enable = TRUE
		BackUp.DataAction = eWrite
		BackUp.DataLength = Backup[n].DataLength
		BackUp.MemType = Backup[n].MemTyp
		BackUp.pData = Backup[n].pData
		BackUp.pFileName = Backup[n].pFileName
		BackUp FUB DataBackUp()
		IF ((BackUp.Status = ERR_OK) OR (BackUp.Status <> ERR_FUB_BUSY)) THEN
			Backup[n].ident = BackUp.CurrentDatFile.ident
			IF (D[myMonitorReg] > 0) THEN
				INC n
				IF (n > MaxBackUpAreas)THEN
					n = 0
					eBackup = eCopyToUSB
				ENDIF
				IF (BackUp.Status = ERR_OK) THEN
					INC Debug.WriteCount_MEM
				ELSE IF (BackUp.Status <> ERR_FUB_BUSY) THEN
					INC Debug.WriteFail_MEM
				ENDIF
			ELSE
				eBackup = eNull
			ENDIF
		ENDIF
	ENDACTION

	ACTION eRead: ; Restore perm memory

		BackUp.Enable = TRUE
		BackUp.DataAction = eRead
		BackUp.DataLength = Backup[n].DataLength
		BackUp.pData = Backup[n].pData
		BackUp.pFileName = Backup[n].pFileName
		BackUp FUB DataBackUp()
		IF ((BackUp.Status = ERR_OK) OR (BackUp.Status <> ERR_FUB_BUSY)) THEN
			Backup[n].ident = BackUp.CurrentDatFile.ident
			INC n
			IF (BackUp.Status = ERR_OK) THEN
				INC Debug.ReadCount_MEM
			ELSE IF (BackUp.Status <> ERR_FUB_BUSY) THEN
				INC Debug.ReadFail_MEM
			ENDIF
			IF (n > MaxBackUpAreas)THEN
				D[myUpdateReg] = 0
				eBackup = eNull
			ENDIF
		ENDIF
	ENDACTION

	ACTION eCopyToUSB: ; Copy all data files to USBStick
		CopytoUSB.Enable = TRUE
		CopytoUSB.pDevice = pUSBDevice
		CopytoUSB.pData = Backup[n].pData
		CopytoUSB.fiLen = Backup[n].DataLength
		CopytoUSB.pFile = Backup[n].pFileName
		CopytoUSB FUB CopyToFileDevice()
		IF CopytoUSB.Status = ERR_OK THEN
			IF (D[myMonitorReg] > 0) THEN
				INC n
				INC Debug.WriteCount_USB
				IF (n > MaxBackUpAreas)THEN
					eBackup = eNull
				ENDIF
			ELSE
				eBackup = eNull
			ENDIF
		ELSE IF CopytoUSB.Status = fiERR_FILE_DEVICE THEN ; File Device doesn't exist go back to writing to SYSROM
			eBackup = eNull
		ELSE IF CopytoUSB.Status <> ERR_FUB_BUSY THEN
			IF (D[myMonitorReg] > 0) THEN
				INC n
				INC Debug.WriteFail_USB
				IF (n > MaxBackUpAreas)THEN
					eBackup = eNull
				ENDIF
			ELSE
				eBackup = eNull
			ENDIF
		ENDIF
	ENDACTION

	ACTION eReadFromUSB:
		ReadFromUSB.Enable = TRUE
		ReadFromUSB.pDevice = pUSBDevice
		ReadFromUSB.pFile = Backup[n].pFileName
		ReadFromUSB.fiLen = Backup[n].DataLength
		ReadFromUSB.pDest = Backup[n].pData
		ReadFromUSB FUB	ReadFromFileDevice()
		IF ReadFromUSB.Status = ERR_OK THEN
			INC n
			INC Debug.ReadCount_USB
			IF (n > MaxBackUpAreas)THEN
				eBackup = eNull
			ENDIF
		ELSE IF ReadFromUSB.Status = fiERR_FILE_DEVICE THEN ; File Device doesn't exist go back to writing to SYSROM
			eBackup = eNull
		ELSE IF  ReadFromUSB.Status <> ERR_FUB_BUSY THEN
			INC n
			INC Debug.ReadFail_USB
			IF (n > MaxBackUpAreas)THEN
				eBackup = eNull
			ENDIF
		ENDIF
	ENDACTION
ENDCASE

IF D[myMonitorReg] = 0 THEN
	Alarm[myAlarm].Name = almBackUpNotRunning
	Alarm[myAlarm].On = TRUE
ENDIF

END_PROGRAM

PROGRAM _EXIT
;Copy all back up files to MemCard

END_PROGRAM
```

### Library Logical/Data_BackUp/DataBackUp (IEC) - *BackUp and Restore Function
Depends on: DataObj

### Package Logical/Robo_Drive_Control - Supertrack Robo Drive Control Package

- Library Logical/Robo_Drive_Control/FC302 (IEC) - FC302 Functions Library (no source held here)

### Package Logical/Robo_Drive_Control/Paramaters_AnaloguePTC - *New parameter lists, for modified PTC wiring

### Data object Logical/Robo_Drive_Control/Paramaters_AnaloguePTC/Param_3kw (Simple, version 4.00.0) - Parameters 3kW Star from Expo Analogue PTC

#### Param_3kw.dat
```
(********************************************************************
 * COPYRIGHT --
 ********************************************************************
 * Data object: Param_2kwStar
 * File: Param_2kwStar.dat
 * Author:  D.Jefferys
 * Created: February 12, 2009
 ********************************************************************
 * Data object file: Param_2kwStar.dat
 ********************************************************************)

;Version 4.01 18/12/2012 T.R. Created 3kw instance based on 2.2kw version 4.00
;CAN Module Switch Settings
;--------------------------

;Baudrate
;8 on  7 on  Par 10-01
;8 on  7 off 500kbps
;8 off 7 on  250kbps
;8 off 7 off 125kbps

;Node Number Binary
;1 = 1s
;2 = 2s
;3 = 4s
;4 = 8s
;5 = 16s
;6 = 32s

;
;	!!! DO NOT CHANGE THE SEQUENCE OF THE PARAMETERS
;
; FU parameter to the Ubertragung (only parameter, which deviates from the default values)
;
; 3 kW Star
;
; Index, Subindex, Datatype (Bytes), Setting (DINT) ; Comments
0002,00,01,00000001	; [000] 00-02, Motor Speed 0 - RPM, 1 - Hz
0001,00,01,00000000	; [001] 00-01, Language 0 - English, 1 - German
0011,00,01,00000001	; [002] 00-11, Edit Setup 1
0190,00,01,00000002	; [003] 01-90, Motor Thermal Protection, 2 - Thermistor
0040,00,01,00000000 ; [004] 00-40, Hand On Key on LCP 0 - Disabled No Function
0381,00,04,00000020 ; [005] 03-81, QuickStop ramp time 100 - 1s
0458,00,01,00000001	; [006] 04-58, Missing motor phase function, 1 - Trip 100ms
0854,00,01,00000001	; [007] 08-54, Reversing select 1 - Bus only 3 - Bus and Terminal
0211,00,02,00000300	; [008] 02-11, Brake resistor 100 Ohm
0212,00,04,00001500	; [009] 02-12, Brake power limit 200 Watt
0213,00,01,00000002	; [010] 02-13, Brake check 2 - Alarm
1426,00,01,00000000 ; [011] 14-26, Trip delay at inverter fault 0 = Disabled
0803,00,04,00000002 ; [012] 08-03, Control Word Timeout Time 10 = 1Sec
0804,00,01,00000002	; [013] 08-04, Control Word Timeout Function 2 - Stop with auto restart
0801,00,01,00000000	; [014] 08-01, Control Site, 0 - Controlword & digital only
0223,00,01,00000005	; [015] 02-23, Active brake delay 0,3 s
1761,00,01,00000002	; [016] 17-61, Encoder Signal Monitoring (Encoder faulty), 2 - Trip
1710,00,01,00000001	; [017] 17-10, Encoder Signal Type 1 - TTL
1711,00,02,00001024	; [018] 17-11, Encoder Resolution 1024 Pulse
0430,00,01,00000001 ; [019] 04-30, Motor Feedback Loss Function, 1 - Warning, 2* - Trip
0431,00,02,00000300 ; [020] 04-31, Motor Feedback Speed Error RPM, 0-600, 300*
0226,00,02,00005000	; [021] 02-26, Torque Ref, 50,00%
0228,00,02,00000200	; [022] 02-28, Gain Boost Factor, 2,00% 0-4% ***************************
0519,00,01,00000003	; [023] 05-19, Terminal 37 Safe Stop, 3 - Safe Stop Warning
0120,00,04,00000300	; [024] 01-20, Motor Power 3kW
0101,00,01,00000003	; [025] 01-01, Motor Control Principle, 3 - Flux with motor feedback
0122,00,02,00000400	; [026] 01-22, Motor voltage 400 V
0123,00,02,00000050	; [027] 01-23, Motor frequency 50 Hz
0162,00,02,00000100	; [028] 01-62, Slip compenstation 100%
0410,00,01,00000002	; [029] 04-10, Motor speed direction, 2 - both directions
0540,00,01,00000032	; [030] 05-40, [0] Relay 1 Function, 32 - Mech brake ctrl
0540,01,01,00000032	; [031] 05-40, [1] Relay 2 Function, 32 - Mech brake ctrl
0802,00,01,00000003 ; [032] 08-02, Control Site 3 - Option A CAN Bus
0102,00,01,00000002	; [033] 01-02, Flux Motor Feeback Source 2 - MCB102
0125,00,02,00001420	; [034] 01-25, Motor nominal speed 1420 rpm
0702,00,02,00000070	; [035] 07-02, Speed PID proportionl gain 0,070
0700,00,01,00000002	; [036] 07-00, Speed PID Feedback Source 2 - MCB102
0172,00,01,00000006	; [037] 01-72, Start function, 6 - Hoist Mech. Brake Rel
0210,00,01,00000001	; [038] 02-10, Brake Function, 1 - Resistor brake
1410,00,01,00000005	; [039] 14-10, Mains failure, 3 - Coasting 5 - Kenetic backup , trip
0193,00,01,00000002	; [040] 01-93, Thermistor source, 2 Analogue input 54 Source terminal 50 for 10V //6 - Digital Input 33
0100,00,01,00000001	; [041] 01-00, Configuration mode, 1 - Closed loop with encoder
0139,00,01,00000004	; [042] 01-39, Motor poles, 4
0511,00,01,00000000	; [043] 05-11, Terminal 19, 0 - No Operation
0512,00,01,00000000	; [044] 05-12, Terminal 27, 0 - No Operation
0513,00,01,00000000	; [045] 05-13, Terminal 29, 0 - No Operation
0514,00,01,00000004	; [046] 05-14, Terminal 32, 4 - Quick Stop
0510,00,01,00000000	; [047] 05-10, Terminal 18, 0 - No Operation
0175,00,02,00000015	; [048] 01-75, Start Speed, 1,5 Hz
0222,00,02,00000005	; [049] 02-22, Activate Brake Speed ?en bei 0,5 Hz
0124,00,04,00000750	; [050] 01-24, Motor current 7.5 A
0341,00,04,00000100	; [051] 03-41, Ramp 1 ramp up time (1 Sec to 50 Hz)
0342,00,04,00000100	; [052] 03-42, Ramp 1 ramp down time (1 Sec to  0 Hz)
0414,00,02,00001000	; [053] 04-14, Motor Speed High Limit 100,0 Hz
0220,00,04,00000260	; [054] 02-20, Release brake current 2,6 A
(*0130,00,04,00029763	; [---] 01-30, Stator resistance (Rs) 2,9763 Ohm
0131,00,04,00022212	; [---] 01-31, Rotor resistance (Rr) 2,2212 Ohm*)
(*0134,00,04,00031036	; [---] 01-34, Rotor leakage reactance (X2) 3,1036 Ohm*)
;0136,00,04,01803904	; [---] 01-36, Iron loss resistance (Rfe) 1803,904 Ohm
;0135,00,04,00653996	; [---] 01-35, Main reactance (Xh) 65,3996 Ohm
0416,00,02,00002500	; [055] 04-16, Torque limit motor mode, 160,0 - % NOW 250%
0417,00,02,00001600	; [056] 04-17, Torque limit generator mode, 160,0 %
;0133,00,04,00031036	; [---] 01-33, Stator leakage reactance (X1), 3,1036 Ohm
0303,00,04,00100000	; [057] 03-03, Maximum Reference, 100,000
0418,00,04,00002100	; [058] 04-18, Current Limit 172,0 % - NOW 210%
0851,00,01,00000003	; [0] 08-51, Quick stop Logical OR
```

### Data object Logical/Robo_Drive_Control/Paramaters_AnaloguePTC/Param_1_5kwStar (Simple, version 4.00.0) - Parameters 1.5kW Star Analogue PTC
